LIN {X 0,Y 452.9,Z 249.571,A -85,B 0,C 180,E1 -8543.803,E2 -8543.803} C_VEL
LIN {X 0,Y 449.955,Z 249.94,A -85,B 0,C 180,E1 -8545.004,E2 -8545.004} C_VEL
LIN {X 0,Y 447.53,Z 250.24,A -85,B 0,C 180,E1 -8545.974,E2 -8545.974} C_VEL
LIN {X 0,Y 446.587,Z 250.358,A -85,B 0,C 180,E1 -8546.724,E2 -8546.724} C_VEL
LIN {X 0,Y 446.562,Z 250.36,A -85,B 0,C 180,E1 -8546.978,E2 -8546.978} C_VEL
LIN {X 0,Y 446.726,Z 250.339,A -85,B 0,C 180,E1 -8550,E2 -8550} C_VEL
LIN {X 0,Y 446.651,Z 250.351,A -85,B 0,C 180,E1 -8552.706,E2 -8552.706} C_VEL
LIN {X 0,Y 446.596,Z 250.356,A -85,B 0,C 180,E1 -8556.324,E2 -8556.324} C_VEL
LIN {X 0,Y 446.495,Z 250.369,A -85,B 0,C 180,E1 -8559.056,E2 -8559.056} C_VEL
LIN {X 0,Y 446.47,Z 250.374,A -85,B 0,C 180,E1 -8562.731,E2 -8562.731} C_VEL
LIN {X 0,Y 446.454,Z 250.374,A -85,B 0,C 180,E1 -8566.24,E2 -8566.24} C_VEL
LIN {X 0,Y 446.408,Z 250.374,A -85,B 0,C 180,E1 -8569.305,E2 -8569.305} C_VEL
LIN {X 0,Y 446.382,Z 250.382,A -85,B 0,C 180,E1 -8572.201,E2 -8572.201} C_VEL
LIN {X 0,Y 446.414,Z 250.374,A -85,B 0,C 180,E1 -8575.154,E2 -8575.154} C_VEL
LIN {X 0,Y 446.425,Z 250.378,A -85,B 0,C 180,E1 -8578.182,E2 -8578.182} C_VEL
LIN {X 0,Y 446.361,Z 250.38,A -85,B 0,C 180,E1 -8581.304,E2 -8581.304} C_VEL
LIN {X 0,Y 446.374,Z 250.381,A -85,B 0,C 180,E1 -8584.527,E2 -8584.527} C_VEL
LIN {X 0,Y 446.387,Z 250.384,A -85,B 0,C 180,E1 -8588.088,E2 -8588.088} C_VEL
LIN {X 0,Y 446.396,Z 250.376,A -85,B 0,C 180,E1 -8590.925,E2 -8590.925} C_VEL
LIN {X 0,Y 446.398,Z 250.383,A -85,B 0,C 180,E1 -8593.845,E2 -8593.845} C_VEL
LIN {X 0,Y 446.432,Z 250.373,A -85,B 0,C 180,E1 -8596.397,E2 -8596.397} C_VEL
LIN {X 0,Y 446.423,Z 250.38,A -85,B 0,C 180,E1 -8599.81,E2 -8599.81} C_VEL
LIN {X 0,Y 446.389,Z 250.379,A -85,B 0,C 180,E1 -8602.129,E2 -8602.129} C_VEL
LIN {X 0,Y 446.391,Z 250.382,A -85,B 0,C 180,E1 -8605.482,E2 -8605.482} C_VEL
LIN {X 0,Y 446.378,Z 250.378,A -85,B 0,C 180,E1 -8608.705,E2 -8608.705} C_VEL
LIN {X 0,Y 446.451,Z 250.372,A -85,B 0,C 180,E1 -8611.827,E2 -8611.827} C_VEL
LIN {X 0,Y 446.418,Z 250.375,A -85,B 0,C 180,E1 -8614.853,E2 -8614.853} C_VEL
LIN {X 0,Y 446.42,Z 250.373,A -85,B 0,C 180,E1 -8618.251,E2 -8618.251} C_VEL
LIN {X 0,Y 446.426,Z 250.374,A -85,B 0,C 180,E1 -8621.655,E2 -8621.655} C_VEL
LIN {X 0,Y 446.485,Z 250.365,A -85,B 0,C 180,E1 -8624.485,E2 -8624.485} C_VEL
LIN {X 0,Y 446.498,Z 250.363,A -85,B 0,C 180,E1 -8628.199,E2 -8628.199} C_VEL
LIN {X 0,Y 446.514,Z 250.368,A -85,B 0,C 180,E1 -8630.95,E2 -8630.95} C_VEL
LIN {X 0,Y 446.612,Z 250.349,A -85,B 0,C 180,E1 -8633.682,E2 -8633.682} C_VEL
LIN {X 0,Y 446.675,Z 250.343,A -85,B 0,C 180,E1 -8637.3,E2 -8637.3} C_VEL
LIN {X 0,Y 446.777,Z 250.329,A -85,B 0,C 180,E1 -8640.005,E2 -8640.005} C_VEL
LIN {X 0,Y 446.652,Z 250.352,A -85,B 0,C 180,E1 -8642.711,E2 -8642.711} C_VEL
LIN {X 0,Y 446.619,Z 250.352,A -85,B 0,C 180,E1 -8646.329,E2 -8646.329} C_VEL
LIN {X 0,Y 446.522,Z 250.362,A -85,B 0,C 180,E1 -8649.06,E2 -8649.06} C_VEL
LIN {X 0,Y 446.519,Z 250.364,A -85,B 0,C 180,E1 -8652.734,E2 -8652.734} C_VEL
LIN {X 0,Y 446.488,Z 250.371,A -85,B 0,C 180,E1 -8656.464,E2 -8656.464} C_VEL
LIN {X 0,Y 446.469,Z 250.367,A -85,B 0,C 180,E1 -8659.308,E2 -8659.308} C_VEL
LIN {X 0,Y 446.42,Z 250.381,A -85,B 0,C 180,E1 -8662.204,E2 -8662.204} C_VEL
LIN {X 0,Y 446.44,Z 250.37,A -85,B 0,C 180,E1 -8665.157,E2 -8665.157} C_VEL
LIN {X 0,Y 446.442,Z 250.376,A -85,B 0,C 180,E1 -8668.186,E2 -8668.186} C_VEL
LIN {X 0,Y 446.42,Z 250.373,A -85,B 0,C 180,E1 -8671.304,E2 -8671.304} C_VEL
LIN {X 0,Y 446.428,Z 250.375,A -85,B 0,C 180,E1 -8674.527,E2 -8674.527} C_VEL
LIN {X 0,Y 446.416,Z 250.38,A -85,B 0,C 180,E1 -8678.081,E2 -8678.081} C_VEL
LIN {X 0,Y 446.426,Z 250.478,A -85,B 0,C 180,E1 -8680.919,E2 -8680.919} C_VEL
LIN {X 0,Y 446.852,Z 253.496,A -85,B 0,C 180,E1 -8683.794,E2 -8683.794} C_VEL
LIN {X 0,Y 447.237,Z 256.331,A -85,B 0,C 180,E1 -8686.295,E2 -8686.295} C_VEL
LIN {X 0,Y 447.28,Z 259.62,A -85,B 0,C 180,E1 -8688.96,E2 -8688.96} C_VEL
LIN {X 0,Y 447.05,Z 263.911,A -85,B 0,C 180,E1 -8692.186,E2 -8692.186} C_VEL
LIN {X 0,Y 446.758,Z 268.648,A -85,B 0,C 180,E1 -8695.507,E2 -8695.507} C_VEL
LIN {X 0,Y 446.52,Z 272.71,A -85,B 0,C 180,E1 -8698.209,E2 -8698.209} C_VEL
LIN {X 0,Y 446.246,Z 276.741,A -85,B 0,C 180,E1 -8700.777,E2 -8700.777} C_VEL
LIN {X 0,Y 445.992,Z 281.876,A -85,B 0,C 180,E1 -8703.929,E2 -8703.929} C_VEL
LIN {X 0,Y 445.81,Z 286.721,A -85,B 0,C 180,E1 -8706.79,E2 -8706.79} C_VEL
LIN {X 0,Y 445.651,Z 291.794,A -85,B 0,C 180,E1 -8709.7,E2 -8709.7} C_VEL
LIN {X 0,Y 445.522,Z 296.887,A -85,B 0,C 180,E1 -8712.56,E2 -8712.56} C_VEL
LIN {X 0,Y 445.488,Z 299.321,A -85,B 0,C 180,E1 -8713.877,E2 -8713.877} C_VEL
LIN {X 0,Y 447.434,Z 310.041,A -85,B 0,C 180,E1 -8714.251,E2 -8714.251} C_VEL
LIN {X 0,Y 448.961,Z 320.875,A -85,B 0,C 180,E1 -8714.741,E2 -8714.741} C_VEL
LIN {X 0,Y 449.114,Z 325.65,A -85,B 0,C 180,E1 -8714.979,E2 -8714.979} C_VEL
LIN {X 0,Y 448.597,Z 336.174,A -85,B 0,C 180,E1 -8715.599,E2 -8715.599} C_VEL
LIN {X 0,Y 448.082,Z 345.452,A -85,B 0,C 180,E1 -8716.277,E2 -8716.277} C_VEL
LIN {X 0,Y 447.587,Z 354.692,A -85,B 0,C 180,E1 -8717.101,E2 -8717.101} C_VEL
LIN {X 0,Y 447.156,Z 362.932,A -85,B 0,C 180,E1 -8717.98,E2 -8717.98} C_VEL
LIN {X 0,Y 446.705,Z 370.151,A -85,B 0,C 180,E1 -8718.888,E2 -8718.888} C_VEL
LIN {X 0,Y 446.388,Z 376.355,A -85,B 0,C 180,E1 -8719.798,E2 -8719.798} C_VEL
LIN {X 0,Y 446.007,Z 382.892,A -85,B 0,C 180,E1 -8720.934,E2 -8720.934} C_VEL
LIN {X 0,Y 445.798,Z 387.393,A -85,B 0,C 180,E1 -8721.843,E2 -8721.843} C_VEL
LIN {X 0,Y 445.57,Z 393.039,A -85,B 0,C 180,E1 -8723.252,E2 -8723.252} C_VEL
LIN {X 0,Y 445.484,Z 397.207,A -85,B 0,C 180,E1 -8724.569,E2 -8724.569} C_VEL
LIN {X 0,Y 445.418,Z 399.572,A -85,B 0,C 180,E1 -8725.475,E2 -8725.475} C_VEL
LIN {X 0,Y 445.432,Z 402.755,A -85,B 0,C 180,E1 -8727.287,E2 -8727.287} C_VEL
LIN {X 0,Y 445.36,Z 403.81,A -85,B 0,C 180,E1 -8728.191,E2 -8728.191} C_VEL
LIN {X 0,Y 445.32,Z 404.396,A -85,B 0,C 180,E1 -8729.096,E2 -8729.096} C_VEL
LIN {X 0,Y 445.32,Z 404.396,A -85,B 0,C 180,E1 -8730.904,E2 -8730.904} C_VEL
LIN {X 0,Y 445.36,Z 403.81,A -85,B 0,C 180,E1 -8731.809,E2 -8731.809} C_VEL
LIN {X 0,Y 445.432,Z 402.755,A -85,B 0,C 180,E1 -8732.713,E2 -8732.713} C_VEL
LIN {X 0,Y 445.418,Z 399.572,A -85,B 0,C 180,E1 -8734.525,E2 -8734.525} C_VEL
LIN {X 0,Y 445.479,Z 395.461,A -85,B 0,C 180,E1 -8736.04,E2 -8736.04} C_VEL
LIN {X 0,Y 445.645,Z 391.224,A -85,B 0,C 180,E1 -8737.248,E2 -8737.248} C_VEL
LIN {X 0,Y 445.898,Z 385.203,A -85,B 0,C 180,E1 -8738.611,E2 -8738.611} C_VEL
LIN {X 0,Y 446.224,Z 379.107,A -85,B 0,C 180,E1 -8739.748,E2 -8739.748} C_VEL
LIN {X 0,Y 446.514,Z 373.405,A -85,B 0,C 180,E1 -8740.657,E2 -8740.657} C_VEL
LIN {X 0,Y 447.055,Z 364.852,A -85,B 0,C 180,E1 -8741.792,E2 -8741.792} C_VEL
LIN {X 0,Y 447.501,Z 356.67,A -85,B 0,C 180,E1 -8742.701,E2 -8742.701} C_VEL
LIN {X 0,Y 447.882,Z 348.534,A -85,B 0,C 180,E1 -8743.465,E2 -8743.465} C_VEL
LIN {X 0,Y 448.429,Z 339.439,A -85,B 0,C 180,E1 -8744.175,E2 -8744.175} C_VEL
LIN {X 0,Y 448.866,Z 330.686,A -85,B 0,C 180,E1 -8744.739,E2 -8744.739} C_VEL
LIN {X 0,Y 449.138,Z 322.169,A -85,B 0,C 180,E1 -8745.194,E2 -8745.194} C_VEL
LIN {X 0,Y 447.538,Z 310.77,A -85,B 0,C 180,E1 -8745.721,E2 -8745.721} C_VEL
LIN {X 0,Y 445.564,Z 300.178,A -85,B 0,C 180,E1 -8746.1,E2 -8746.1} C_VEL
LIN {X 0,Y 445.489,Z 299.318,A -85,B 0,C 180,E1 -8746.125,E2 -8746.125} C_VEL
LIN {X 0,Y 445.615,Z 293.467,A -85,B 0,C 180,E1 -8749.341,E2 -8749.341} C_VEL
LIN {X 0,Y 445.743,Z 288.39,A -85,B 0,C 180,E1 -8752.234,E2 -8752.234} C_VEL
LIN {X 0,Y 445.92,Z 283.357,A -85,B 0,C 180,E1 -8755.184,E2 -8755.184} C_VEL
LIN {X 0,Y 446.157,Z 278.379,A -85,B 0,C 180,E1 -8758.2,E2 -8758.2} C_VEL
LIN {X 0,Y 446.468,Z 273.469,A -85,B 0,C 180,E1 -8761.295,E2 -8761.295} C_VEL
LIN {X 0,Y 446.768,Z 268.64,A -85,B 0,C 180,E1 -8764.492,E2 -8764.492} C_VEL
LIN {X 0,Y 447.032,Z 263.899,A -85,B 0,C 180,E1 -8767.816,E2 -8767.816} C_VEL
LIN {X 0,Y 447.192,Z 260.798,A -85,B 0,C 180,E1 -8770.116,E2 -8770.116} C_VEL
LIN {X 0,Y 447.312,Z 257.769,A -85,B 0,C 180,E1 -8772.499,E2 -8772.499} C_VEL
LIN {X 0,Y 447.06,Z 254.794,A -85,B 0,C 180,E1 -8775.024,E2 -8775.024} C_VEL
LIN {X 0,Y 446.503,Z 250.948,A -85,B 0,C 180,E1 -8778.614,E2 -8778.614} C_VEL
LIN {X 0,Y 446.426,Z 250.477,A -85,B 0,C 180,E1 -8779.081,E2 -8779.081} C_VEL
LIN {X 0,Y 446.41,Z 250.382,A -85,B 0,C 180,E1 -8782.117,E2 -8782.117} C_VEL
LIN {X 0,Y 446.428,Z 250.378,A -85,B 0,C 180,E1 -8785.473,E2 -8785.473} C_VEL
LIN {X 0,Y 446.42,Z 250.373,A -85,B 0,C 180,E1 -8788.696,E2 -8788.696} C_VEL
LIN {X 0,Y 446.451,Z 250.375,A -85,B 0,C 180,E1 -8791.827,E2 -8791.827} C_VEL
LIN {X 0,Y 446.44,Z 250.37,A -85,B 0,C 180,E1 -8794.843,E2 -8794.843} C_VEL
LIN {X 0,Y 446.45,Z 250.371,A -85,B 0,C 180,E1 -8798.241,E2 -8798.241} C_VEL
LIN {X 0,Y 446.451,Z 250.376,A -85,B 0,C 180,E1 -8801.645,E2 -8801.645} C_VEL
LIN {X 0,Y 446.506,Z 250.362,A -85,B 0,C 180,E1 -8804.475,E2 -8804.475} C_VEL
LIN {X 0,Y 446.513,Z 250.362,A -85,B 0,C 180,E1 -8808.188,E2 -8808.188} C_VEL
LIN {X 0,Y 446.522,Z 250.362,A -85,B 0,C 180,E1 -8810.94,E2 -8810.94} C_VEL
LIN {X 0,Y 446.619,Z 250.352,A -85,B 0,C 180,E1 -8813.671,E2 -8813.671} C_VEL
LIN {X 0,Y 446.652,Z 250.352,A -85,B 0,C 180,E1 -8817.289,E2 -8817.289} C_VEL
LIN {X 0,Y 446.777,Z 250.329,A -85,B 0,C 180,E1 -8819.995,E2 -8819.995} C_VEL
LIN {X 0,Y 446.675,Z 250.343,A -85,B 0,C 180,E1 -8822.7,E2 -8822.7} C_VEL
LIN {X 0,Y 446.612,Z 250.349,A -85,B 0,C 180,E1 -8826.318,E2 -8826.318} C_VEL
LIN {X 0,Y 446.514,Z 250.368,A -85,B 0,C 180,E1 -8829.05,E2 -8829.05} C_VEL
LIN {X 0,Y 446.501,Z 250.368,A -85,B 0,C 180,E1 -8832.724,E2 -8832.724} C_VEL
LIN {X 0,Y 446.472,Z 250.367,A -85,B 0,C 180,E1 -8836.222,E2 -8836.222} C_VEL
LIN {X 0,Y 446.442,Z 250.372,A -85,B 0,C 180,E1 -8839.298,E2 -8839.298} C_VEL
LIN {X 0,Y 446.389,Z 250.379,A -85,B 0,C 180,E1 -8842.194,E2 -8842.194} C_VEL
LIN {X 0,Y 446.418,Z 250.375,A -85,B 0,C 180,E1 -8845.147,E2 -8845.147} C_VEL
LIN {X 0,Y 446.451,Z 250.372,A -85,B 0,C 180,E1 -8848.173,E2 -8848.173} C_VEL
LIN {X 0,Y 446.381,Z 250.378,A -85,B 0,C 180,E1 -8851.769,E2 -8851.769} C_VEL
LIN {X 0,Y 446.391,Z 250.382,A -85,B 0,C 180,E1 -8854.518,E2 -8854.518} C_VEL
LIN {X 0,Y 446.392,Z 250.381,A -85,B 0,C 180,E1 -8858.077,E2 -8858.077} C_VEL
LIN {X 0,Y 446.403,Z 250.376,A -85,B 0,C 180,E1 -8860.916,E2 -8860.916} C_VEL
LIN {X 0,Y 446.432,Z 250.375,A -85,B 0,C 180,E1 -8863.831,E2 -8863.831} C_VEL
LIN {X 0,Y 446.4,Z 250.376,A -85,B 0,C 180,E1 -8867.393,E2 -8867.393} C_VEL
LIN {X 0,Y 446.444,Z 250.372,A -85,B 0,C 180,E1 -8870.464,E2 -8870.464} C_VEL
LIN {X 0,Y 446.353,Z 250.383,A -85,B 0,C 180,E1 -8873.405,E2 -8873.405} C_VEL
LIN {X 0,Y 446.392,Z 250.377,A -85,B 0,C 180,E1 -8876.563,E2 -8876.563} C_VEL
LIN {X 0,Y 446.382,Z 250.382,A -85,B 0,C 180,E1 -8879.973,E2 -8879.973} C_VEL
LIN {X 0,Y 446.422,Z 250.373,A -85,B 0,C 180,E1 -8882.836,E2 -8882.836} C_VEL
LIN {X 0,Y 446.411,Z 250.378,A -85,B 0,C 180,E1 -8885.918,E2 -8885.918} C_VEL
LIN {X 0,Y 446.433,Z 250.372,A -85,B 0,C 180,E1 -8888.773,E2 -8888.773} C_VEL
LIN {X 0,Y 446.401,Z 250.382,A -85,B 0,C 180,E1 -8891.647,E2 -8891.647} C_VEL
LIN {X 0,Y 446.462,Z 250.371,A -85,B 0,C 180,E1 -8894.479,E2 -8894.479} C_VEL
LIN {X 0,Y 446.481,Z 250.368,A -85,B 0,C 180,E1 -8898.192,E2 -8898.192} C_VEL
LIN {X 0,Y 446.54,Z 250.362,A -85,B 0,C 180,E1 -8901.857,E2 -8901.857} C_VEL
LIN {X 0,Y 446.591,Z 250.356,A -85,B 0,C 180,E1 -8904.582,E2 -8904.582} C_VEL
LIN {X 0,Y 446.562,Z 250.36,A -85,B 0,C 180,E1 -8906.978,E2 -8906.978} C_VEL
LIN {X 0,Y 446.044,Z 250.428,A -85,B 0,C 180,E1 -8907.731,E2 -8907.731} C_VEL
LIN {X 0,Y 443.253,Z 250.781,A -85,B 0,C 180,E1 -8908.955,E2 -8908.955} C_VEL
LIN {X 0,Y 440.784,Z 251.087,A -85,B 0,C 180,E1 -8909.942,E2 -8909.942} C_VEL
LIN {X 0,Y 439.689,Z 251.219,A -85,B 0,C 180,E1 -8910.705,E2 -8910.705} C_VEL
LIN {X 0,Y 439.587,Z 251.23,A -85,B 0,C 180,E1 -8910.964,E2 -8910.964} C_VEL
LIN {X 0,Y 439.599,Z 251.229,A -85,B 0,C 180,E1 -8912.749,E2 -8912.749} C_VEL
LIN {X 0,Y 439.566,Z 251.233,A -85,B 0,C 180,E1 -8916.426,E2 -8916.426} C_VEL
LIN {X 0,Y 439.452,Z 251.246,A -85,B 0,C 180,E1 -8919.202,E2 -8919.202} C_VEL
LIN {X 0,Y 439.439,Z 251.25,A -85,B 0,C 180,E1 -8922.728,E2 -8922.728} C_VEL
LIN {X 0,Y 439.397,Z 251.254,A -85,B 0,C 180,E1 -8926.357,E2 -8926.357} C_VEL
LIN {X 0,Y 439.373,Z 251.252,A -85,B 0,C 180,E1 -8929.627,E2 -8929.627} C_VEL
LIN {X 0,Y 439.324,Z 251.263,A -85,B 0,C 180,E1 -8932.577,E2 -8932.577} C_VEL
LIN {X 0,Y 439.354,Z 251.253,A -85,B 0,C 180,E1 -8935.587,E2 -8935.587} C_VEL
LIN {X 0,Y 439.366,Z 251.254,A -85,B 0,C 180,E1 -8938.676,E2 -8938.676} C_VEL
LIN {X 0,Y 439.316,Z 251.261,A -85,B 0,C 180,E1 -8941.864,E2 -8941.864} C_VEL
LIN {X 0,Y 439.345,Z 251.254,A -85,B 0,C 180,E1 -8945.16,E2 -8945.16} C_VEL
LIN {X 0,Y 439.349,Z 251.255,A -85,B 0,C 180,E1 -8948.597,E2 -8948.597} C_VEL
LIN {X 0,Y 439.354,Z 251.254,A -85,B 0,C 180,E1 -8951.264,E2 -8951.264} C_VEL
LIN {X 0,Y 439.368,Z 251.251,A -85,B 0,C 180,E1 -8954.732,E2 -8954.732} C_VEL
LIN {X 0,Y 439.369,Z 251.259,A -85,B 0,C 180,E1 -8957.803,E2 -8957.803} C_VEL
LIN {X 0,Y 439.405,Z 251.249,A -85,B 0,C 180,E1 -8960.235,E2 -8960.235} C_VEL
LIN {X 0,Y 439.336,Z 251.262,A -85,B 0,C 180,E1 -8963.718,E2 -8963.718} C_VEL
LIN {X 0,Y 439.334,Z 251.257,A -85,B 0,C 180,E1 -8967.059,E2 -8967.059} C_VEL
LIN {X 0,Y 439.346,Z 251.254,A -85,B 0,C 180,E1 -8970.28,E2 -8970.28} C_VEL
LIN {X 0,Y 439.396,Z 251.255,A -85,B 0,C 180,E1 -8973.402,E2 -8973.402} C_VEL
LIN {X 0,Y 439.356,Z 251.253,A -85,B 0,C 180,E1 -8976.435,E2 -8976.435} C_VEL
LIN {X 0,Y 439.361,Z 251.258,A -85,B 0,C 180,E1 -8979.403,E2 -8979.403} C_VEL
LIN {X 0,Y 439.38,Z 251.25,A -85,B 0,C 180,E1 -8982.314,E2 -8982.314} C_VEL
LIN {X 0,Y 439.425,Z 251.251,A -85,B 0,C 180,E1 -8985.18,E2 -8985.18} C_VEL
LIN {X 0,Y 439.464,Z 251.239,A -85,B 0,C 180,E1 -8988.007,E2 -8988.007} C_VEL
LIN {X 0,Y 439.487,Z 251.237,A -85,B 0,C 180,E1 -8991.731,E2 -8991.731} C_VEL
LIN {X 0,Y 439.594,Z 251.226,A -85,B 0,C 180,E1 -8994.501,E2 -8994.501} C_VEL
LIN {X 0,Y 439.622,Z 251.221,A -85,B 0,C 180,E1 -8998.173,E2 -8998.173} C_VEL
LIN {X 0,Y 439.747,Z 251.204,A -85,B 0,C 180,E1 -9000.005,E2 -9000.005} C_VEL
LIN {X 0,Y 439.603,Z 251.229,A -85,B 0,C 180,E1 -9002.754,E2 -9002.754} C_VEL
LIN {X 0,Y 439.59,Z 251.229,A -85,B 0,C 180,E1 -9006.431,E2 -9006.431} C_VEL
LIN {X 0,Y 439.486,Z 251.237,A -85,B 0,C 180,E1 -9009.207,E2 -9009.207} C_VEL
LIN {X 0,Y 439.463,Z 251.241,A -85,B 0,C 180,E1 -9012.942,E2 -9012.942} C_VEL
LIN {X 0,Y 439.445,Z 251.249,A -85,B 0,C 180,E1 -9016.352,E2 -9016.352} C_VEL
LIN {X 0,Y 439.403,Z 251.248,A -85,B 0,C 180,E1 -9019.631,E2 -9019.631} C_VEL
LIN {X 0,Y 439.365,Z 251.255,A -85,B 0,C 180,E1 -9022.58,E2 -9022.58} C_VEL
LIN {X 0,Y 439.378,Z 251.252,A -85,B 0,C 180,E1 -9025.591,E2 -9025.591} C_VEL
LIN {X 0,Y 439.395,Z 251.249,A -85,B 0,C 180,E1 -9028.679,E2 -9028.679} C_VEL
LIN {X 0,Y 439.374,Z 251.257,A -85,B 0,C 180,E1 -9032.033,E2 -9032.033} C_VEL
LIN {X 0,Y 439.396,Z 251.249,A -85,B 0,C 180,E1 -9035.343,E2 -9035.343} C_VEL
LIN {X 0,Y 439.368,Z 251.257,A -85,B 0,C 180,E1 -9038.601,E2 -9038.601} C_VEL
LIN {X 0,Y 439.354,Z 251.26,A -85,B 0,C 180,E1 -9039.843,E2 -9039.843} C_VEL
LIN {X 0,Y 439.491,Z 252.002,A -85,B 0,C 180,E1 -9041.274,E2 -9041.274} C_VEL
LIN {X 0,Y 439.893,Z 254.89,A -85,B 0,C 180,E1 -9044.034,E2 -9044.034} C_VEL
LIN {X 0,Y 440.24,Z 257.847,A -85,B 0,C 180,E1 -9046.651,E2 -9046.651} C_VEL
LIN {X 0,Y 440.236,Z 260.851,A -85,B 0,C 180,E1 -9049.117,E2 -9049.117} C_VEL
LIN {X 0,Y 440.095,Z 263.955,A -85,B 0,C 180,E1 -9051.494,E2 -9051.494} C_VEL
LIN {X 0,Y 439.775,Z 268.634,A -85,B 0,C 180,E1 -9054.88,E2 -9054.88} C_VEL
LIN {X 0,Y 439.476,Z 273.44,A -85,B 0,C 180,E1 -9058.149,E2 -9058.149} C_VEL
LIN {X 0,Y 439.122,Z 278.32,A -85,B 0,C 180,E1 -9061.306,E2 -9061.306} C_VEL
LIN {X 0,Y 438.876,Z 283.271,A -85,B 0,C 180,E1 -9064.383,E2 -9064.383} C_VEL
LIN {X 0,Y 438.677,Z 288.279,A -85,B 0,C 180,E1 -9067.388,E2 -9067.388} C_VEL
LIN {X 0,Y 438.544,Z 293.332,A -85,B 0,C 180,E1 -9070.334,E2 -9070.334} C_VEL
LIN {X 0,Y 438.414,Z 299.15,A -85,B 0,C 180,E1 -9073.608,E2 -9073.608} C_VEL
LIN {X 0,Y 440.551,Z 310.914,A -85,B 0,C 180,E1 -9074.035,E2 -9074.035} C_VEL
LIN {X 0,Y 442.279,Z 323.261,A -85,B 0,C 180,E1 -9074.623,E2 -9074.623} C_VEL
LIN {X 0,Y 441.708,Z 335.979,A -85,B 0,C 180,E1 -9075.37,E2 -9075.37} C_VEL
LIN {X 0,Y 441.176,Z 345.257,A -85,B 0,C 180,E1 -9076.058,E2 -9076.058} C_VEL
LIN {X 0,Y 440.752,Z 353.31,A -85,B 0,C 180,E1 -9076.774,E2 -9076.774} C_VEL
LIN {X 0,Y 440.316,Z 360.817,A -85,B 0,C 180,E1 -9077.557,E2 -9077.557} C_VEL
LIN {X 0,Y 439.723,Z 369.956,A -85,B 0,C 180,E1 -9078.709,E2 -9078.709} C_VEL
LIN {X 0,Y 439.364,Z 376.159,A -85,B 0,C 180,E1 -9079.633,E2 -9079.633} C_VEL
LIN {X 0,Y 438.981,Z 382.697,A -85,B 0,C 180,E1 -9080.788,E2 -9080.788} C_VEL
LIN {X 0,Y 438.751,Z 387.198,A -85,B 0,C 180,E1 -9081.711,E2 -9081.711} C_VEL
LIN {X 0,Y 438.512,Z 392.689,A -85,B 0,C 180,E1 -9083.096,E2 -9083.096} C_VEL
LIN {X 0,Y 438.383,Z 397.012,A -85,B 0,C 180,E1 -9084.48,E2 -9084.48} C_VEL
LIN {X 0,Y 438.348,Z 399.377,A -85,B 0,C 180,E1 -9085.402,E2 -9085.402} C_VEL
LIN {X 0,Y 438.265,Z 401.173,A -85,B 0,C 180,E1 -9086.322,E2 -9086.322} C_VEL
LIN {X 0,Y 438.34,Z 402.561,A -85,B 0,C 180,E1 -9087.243,E2 -9087.243} C_VEL
LIN {X 0,Y 438.283,Z 403.616,A -85,B 0,C 180,E1 -9088.162,E2 -9088.162} C_VEL
LIN {X 0,Y 438.235,Z 404.202,A -85,B 0,C 180,E1 -9089.081,E2 -9089.081} C_VEL
LIN {X 0,Y 438.235,Z 404.202,A -85,B 0,C 180,E1 -9090.919,E2 -9090.919} C_VEL
LIN {X 0,Y 438.283,Z 403.616,A -85,B 0,C 180,E1 -9091.838,E2 -9091.838} C_VEL
LIN {X 0,Y 438.34,Z 402.561,A -85,B 0,C 180,E1 -9092.757,E2 -9092.757} C_VEL
LIN {X 0,Y 438.265,Z 401.173,A -85,B 0,C 180,E1 -9093.678,E2 -9093.678} C_VEL
LIN {X 0,Y 438.389,Z 398.229,A -85,B 0,C 180,E1 -9095.058,E2 -9095.058} C_VEL
LIN {X 0,Y 438.46,Z 394.242,A -85,B 0,C 180,E1 -9096.442,E2 -9096.442} C_VEL
LIN {X 0,Y 438.661,Z 389.114,A -85,B 0,C 180,E1 -9097.827,E2 -9097.827} C_VEL
LIN {X 0,Y 438.9,Z 383.852,A -85,B 0,C 180,E1 -9098.982,E2 -9098.982} C_VEL
LIN {X 0,Y 439.279,Z 377.535,A -85,B 0,C 180,E1 -9100.136,E2 -9100.136} C_VEL
LIN {X 0,Y 439.596,Z 371.583,A -85,B 0,C 180,E1 -9101.06,E2 -9101.06} C_VEL
LIN {X 0,Y 440.078,Z 364.656,A -85,B 0,C 180,E1 -9101.982,E2 -9101.982} C_VEL
LIN {X 0,Y 440.54,Z 356.474,A -85,B 0,C 180,E1 -9102.905,E2 -9102.905} C_VEL
LIN {X 0,Y 440.981,Z 347.693,A -85,B 0,C 180,E1 -9103.736,E2 -9103.736} C_VEL
LIN {X 0,Y 441.506,Z 339.243,A -85,B 0,C 180,E1 -9104.402,E2 -9104.402} C_VEL
LIN {X 0,Y 442.003,Z 330.491,A -85,B 0,C 180,E1 -9104.974,E2 -9104.974} C_VEL
LIN {X 0,Y 442.287,Z 323.262,A -85,B 0,C 180,E1 -9105.376,E2 -9105.376} C_VEL
LIN {X 0,Y 440.606,Z 311.162,A -85,B 0,C 180,E1 -9105.955,E2 -9105.955} C_VEL
LIN {X 0,Y 438.534,Z 300.22,A -85,B 0,C 180,E1 -9106.359,E2 -9106.359} C_VEL
LIN {X 0,Y 438.413,Z 299.149,A -85,B 0,C 180,E1 -9106.393,E2 -9106.393} C_VEL
LIN {X 0,Y 438.543,Z 293.33,A -85,B 0,C 180,E1 -9109.666,E2 -9109.666} C_VEL
LIN {X 0,Y 438.692,Z 288.278,A -85,B 0,C 180,E1 -9112.611,E2 -9112.611} C_VEL
LIN {X 0,Y 438.88,Z 283.27,A -85,B 0,C 180,E1 -9115.617,E2 -9115.617} C_VEL
LIN {X 0,Y 439.121,Z 278.317,A -85,B 0,C 180,E1 -9118.694,E2 -9118.694} C_VEL
LIN {X 0,Y 439.486,Z 273.434,A -85,B 0,C 180,E1 -9121.85,E2 -9121.85} C_VEL
LIN {X 0,Y 439.788,Z 268.625,A -85,B 0,C 180,E1 -9125.119,E2 -9125.119} C_VEL
LIN {X 0,Y 440.072,Z 263.921,A -85,B 0,C 180,E1 -9128.522,E2 -9128.522} C_VEL
LIN {X 0,Y 440.284,Z 260.209,A -85,B 0,C 180,E1 -9131.385,E2 -9131.385} C_VEL
LIN {X 0,Y 440.16,Z 256.981,A -85,B 0,C 180,E1 -9134.064,E2 -9134.064} C_VEL
LIN {X 0,Y 439.71,Z 253.437,A -85,B 0,C 180,E1 -9137.325,E2 -9137.325} C_VEL
LIN {X 0,Y 439.453,Z 251.708,A -85,B 0,C 180,E1 -9139.023,E2 -9139.023} C_VEL
LIN {X 0,Y 439.367,Z 251.258,A -85,B 0,C 180,E1 -9140.217,E2 -9140.217} C_VEL
LIN {X 0,Y 439.377,Z 251.256,A -85,B 0,C 180,E1 -9143.709,E2 -9143.709} C_VEL
LIN {X 0,Y 439.377,Z 251.25,A -85,B 0,C 180,E1 -9147.05,E2 -9147.05} C_VEL
LIN {X 0,Y 439.377,Z 251.254,A -85,B 0,C 180,E1 -9150.27,E2 -9150.27} C_VEL
LIN {X 0,Y 439.373,Z 251.252,A -85,B 0,C 180,E1 -9153.388,E2 -9153.388} C_VEL
LIN {X 0,Y 439.384,Z 251.25,A -85,B 0,C 180,E1 -9156.425,E2 -9156.425} C_VEL
LIN {X 0,Y 439.388,Z 251.252,A -85,B 0,C 180,E1 -9159.393,E2 -9159.393} C_VEL
LIN {X 0,Y 439.403,Z 251.248,A -85,B 0,C 180,E1 -9162.304,E2 -9162.304} C_VEL
LIN {X 0,Y 439.445,Z 251.244,A -85,B 0,C 180,E1 -9165.169,E2 -9165.169} C_VEL
LIN {X 0,Y 439.48,Z 251.24,A -85,B 0,C 180,E1 -9167.996,E2 -9167.996} C_VEL
LIN {X 0,Y 439.497,Z 251.239,A -85,B 0,C 180,E1 -9171.72,E2 -9171.72} C_VEL
LIN {X 0,Y 439.602,Z 251.222,A -85,B 0,C 180,E1 -9174.491,E2 -9174.491} C_VEL
LIN {X 0,Y 439.617,Z 251.22,A -85,B 0,C 180,E1 -9178.163,E2 -9178.163} C_VEL
LIN {X 0,Y 439.747,Z 251.204,A -85,B 0,C 180,E1 -9179.995,E2 -9179.995} C_VEL
LIN {X 0,Y 439.625,Z 251.222,A -85,B 0,C 180,E1 -9182.743,E2 -9182.743} C_VEL
LIN {X 0,Y 439.583,Z 251.225,A -85,B 0,C 180,E1 -9186.42,E2 -9186.42} C_VEL
LIN {X 0,Y 439.477,Z 251.243,A -85,B 0,C 180,E1 -9189.196,E2 -9189.196} C_VEL
LIN {X 0,Y 439.445,Z 251.249,A -85,B 0,C 180,E1 -9192.932,E2 -9192.932} C_VEL
LIN {X 0,Y 439.423,Z 251.246,A -85,B 0,C 180,E1 -9196.342,E2 -9196.342} C_VEL
LIN {X 0,Y 439.376,Z 251.25,A -85,B 0,C 180,E1 -9199.621,E2 -9199.621} C_VEL
LIN {X 0,Y 439.336,Z 251.262,A -85,B 0,C 180,E1 -9202.57,E2 -9202.57} C_VEL
LIN {X 0,Y 439.369,Z 251.251,A -85,B 0,C 180,E1 -9205.58,E2 -9205.58} C_VEL
LIN {X 0,Y 439.383,Z 251.255,A -85,B 0,C 180,E1 -9208.668,E2 -9208.668} C_VEL
LIN {X 0,Y 439.332,Z 251.258,A -85,B 0,C 180,E1 -9212.025,E2 -9212.025} C_VEL
LIN {X 0,Y 439.356,Z 251.253,A -85,B 0,C 180,E1 -9215.335,E2 -9215.335} C_VEL
LIN {X 0,Y 439.352,Z 251.257,A -85,B 0,C 180,E1 -9218.588,E2 -9218.588} C_VEL
LIN {X 0,Y 439.36,Z 251.252,A -85,B 0,C 180,E1 -9221.254,E2 -9221.254} C_VEL
LIN {X 0,Y 439.394,Z 251.249,A -85,B 0,C 180,E1 -9224.719,E2 -9224.719} C_VEL
LIN {X 0,Y 439.362,Z 251.256,A -85,B 0,C 180,E1 -9227.793,E2 -9227.793} C_VEL
LIN {X 0,Y 439.403,Z 251.251,A -85,B 0,C 180,E1 -9230.226,E2 -9230.226} C_VEL
LIN {X 0,Y 439.322,Z 251.262,A -85,B 0,C 180,E1 -9233.709,E2 -9233.709} C_VEL
LIN {X 0,Y 439.316,Z 251.258,A -85,B 0,C 180,E1 -9237.05,E2 -9237.05} C_VEL
LIN {X 0,Y 439.337,Z 251.257,A -85,B 0,C 180,E1 -9240.272,E2 -9240.272} C_VEL
LIN {X 0,Y 439.37,Z 251.255,A -85,B 0,C 180,E1 -9243.393,E2 -9243.393} C_VEL
LIN {X 0,Y 439.339,Z 251.255,A -85,B 0,C 180,E1 -9246.427,E2 -9246.427} C_VEL
LIN {X 0,Y 439.351,Z 251.26,A -85,B 0,C 180,E1 -9249.396,E2 -9249.396} C_VEL
LIN {X 0,Y 439.375,Z 251.254,A -85,B 0,C 180,E1 -9252.308,E2 -9252.308} C_VEL
LIN {X 0,Y 439.399,Z 251.254,A -85,B 0,C 180,E1 -9255.173,E2 -9255.173} C_VEL
LIN {X 0,Y 439.447,Z 251.244,A -85,B 0,C 180,E1 -9258.001,E2 -9258.001} C_VEL
LIN {X 0,Y 439.488,Z 251.241,A -85,B 0,C 180,E1 -9261.725,E2 -9261.725} C_VEL
LIN {X 0,Y 439.566,Z 251.231,A -85,B 0,C 180,E1 -9264.495,E2 -9264.495} C_VEL
LIN {X 0,Y 439.57,Z 251.229,A -85,B 0,C 180,E1 -9268.168,E2 -9268.168} C_VEL
LIN {X 0,Y 439.697,Z 251.215,A -85,B 0,C 180,E1 -9270,E2 -9270} C_VEL
LIN {X 0,Y 439.587,Z 251.23,A -85,B 0,C 180,E1 -9270.964,E2 -9270.964} C_VEL
LIN {X 0,Y 438.85,Z 251.319,A -85,B 0,C 180,E1 -9271.728,E2 -9271.728} C_VEL
LIN {X 0,Y 435.861,Z 251.694,A -85,B 0,C 180,E1 -9272.967,E2 -9272.967} C_VEL
LIN {X 0,Y 433.413,Z 251.999,A -85,B 0,C 180,E1 -9273.967,E2 -9273.967} C_VEL
LIN {X 0,Y 432.442,Z 252.12,A -85,B 0,C 180,E1 -9274.742,E2 -9274.742} C_VEL
LIN {X 0,Y 432.404,Z 252.122,A -85,B 0,C 180,E1 -9275.004,E2 -9275.004} C_VEL
LIN {X 0,Y 432.52,Z 252.109,A -85,B 0,C 180,E1 -9277.68,E2 -9277.68} C_VEL
LIN {X 0,Y 432.35,Z 252.13,A -85,B 0,C 180,E1 -9281.248,E2 -9281.248} C_VEL
LIN {X 0,Y 432.329,Z 252.133,A -85,B 0,C 180,E1 -9284.113,E2 -9284.113} C_VEL
LIN {X 0,Y 432.338,Z 252.133,A -85,B 0,C 180,E1 -9287.014,E2 -9287.014} C_VEL
LIN {X 0,Y 432.32,Z 252.134,A -85,B 0,C 180,E1 -9289.961,E2 -9289.961} C_VEL
LIN {X 0,Y 432.273,Z 252.137,A -85,B 0,C 180,E1 -9292.966,E2 -9292.966} C_VEL
LIN {X 0,Y 432.309,Z 252.134,A -85,B 0,C 180,E1 -9296.035,E2 -9296.035} C_VEL
LIN {X 0,Y 432.294,Z 252.133,A -85,B 0,C 180,E1 -9299.19,E2 -9299.19} C_VEL
LIN {X 0,Y 432.268,Z 252.142,A -85,B 0,C 180,E1 -9302.297,E2 -9302.297} C_VEL
LIN {X 0,Y 432.285,Z 252.135,A -85,B 0,C 180,E1 -9304.681,E2 -9304.681} C_VEL
LIN {X 0,Y 432.302,Z 252.138,A -85,B 0,C 180,E1 -9308.152,E2 -9308.152} C_VEL
LIN {X 0,Y 432.323,Z 252.132,A -85,B 0,C 180,E1 -9311.613,E2 -9311.613} C_VEL
LIN {X 0,Y 432.331,Z 252.13,A -85,B 0,C 180,E1 -9314.346,E2 -9314.346} C_VEL
LIN {X 0,Y 432.327,Z 252.129,A -85,B 0,C 180,E1 -9317.013,E2 -9317.013} C_VEL
LIN {X 0,Y 432.313,Z 252.137,A -85,B 0,C 180,E1 -9319.822,E2 -9319.822} C_VEL
LIN {X 0,Y 432.275,Z 252.136,A -85,B 0,C 180,E1 -9323.028,E2 -9323.028} C_VEL
LIN {X 0,Y 432.321,Z 252.132,A -85,B 0,C 180,E1 -9326.002,E2 -9326.002} C_VEL
LIN {X 0,Y 432.311,Z 252.138,A -85,B 0,C 180,E1 -9329.496,E2 -9329.496} C_VEL
LIN {X 0,Y 432.358,Z 252.126,A -85,B 0,C 180,E1 -9332.934,E2 -9332.934} C_VEL
LIN {X 0,Y 432.34,Z 252.128,A -85,B 0,C 180,E1 -9336.029,E2 -9336.029} C_VEL
LIN {X 0,Y 432.323,Z 252.133,A -85,B 0,C 180,E1 -9339.052,E2 -9339.052} C_VEL
LIN {X 0,Y 432.336,Z 252.128,A -85,B 0,C 180,E1 -9342.016,E2 -9342.016} C_VEL
LIN {X 0,Y 432.372,Z 252.128,A -85,B 0,C 180,E1 -9344.932,E2 -9344.932} C_VEL
LIN {X 0,Y 432.439,Z 252.115,A -85,B 0,C 180,E1 -9347.809,E2 -9347.809} C_VEL
LIN {X 0,Y 432.447,Z 252.114,A -85,B 0,C 180,E1 -9351.595,E2 -9351.595} C_VEL
LIN {X 0,Y 432.571,Z 252.1,A -85,B 0,C 180,E1 -9354.412,E2 -9354.412} C_VEL
LIN {X 0,Y 432.592,Z 252.096,A -85,B 0,C 180,E1 -9358.144,E2 -9358.144} C_VEL
LIN {X 0,Y 432.717,Z 252.08,A -85,B 0,C 180,E1 -9360.005,E2 -9360.005} C_VEL
LIN {X 0,Y 432.557,Z 252.106,A -85,B 0,C 180,E1 -9362.799,E2 -9362.799} C_VEL
LIN {X 0,Y 432.578,Z 252.097,A -85,B 0,C 180,E1 -9365.599,E2 -9365.599} C_VEL
LIN {X 0,Y 432.457,Z 252.118,A -85,B 0,C 180,E1 -9368.415,E2 -9368.415} C_VEL
LIN {X 0,Y 432.456,Z 252.117,A -85,B 0,C 180,E1 -9372.201,E2 -9372.201} C_VEL
LIN {X 0,Y 432.429,Z 252.119,A -85,B 0,C 180,E1 -9376.044,E2 -9376.044} C_VEL
LIN {X 0,Y 432.388,Z 252.121,A -85,B 0,C 180,E1 -9379.489,E2 -9379.489} C_VEL
LIN {X 0,Y 432.319,Z 252.13,A -85,B 0,C 180,E1 -9382.969,E2 -9382.969} C_VEL
LIN {X 0,Y 432.339,Z 252.127,A -85,B 0,C 180,E1 -9385.006,E2 -9385.006} C_VEL
LIN {X 0,Y 432.352,Z 252.127,A -85,B 0,C 180,E1 -9388.626,E2 -9388.626} C_VEL
LIN {X 0,Y 432.325,Z 252.13,A -85,B 0,C 180,E1 -9391.35,E2 -9391.35} C_VEL
LIN {X 0,Y 432.34,Z 252.129,A -85,B 0,C 180,E1 -9394.681,E2 -9394.681} C_VEL
LIN {X 0,Y 432.336,Z 252.134,A -85,B 0,C 180,E1 -9398.154,E2 -9398.154} C_VEL
LIN {X 0,Y 432.317,Z 252.137,A -85,B 0,C 180,E1 -9400.178,E2 -9400.178} C_VEL
LIN {X 0,Y 432.739,Z 254.967,A -85,B 0,C 180,E1 -9403.045,E2 -9403.045} C_VEL
LIN {X 0,Y 433.114,Z 257.899,A -85,B 0,C 180,E1 -9405.755,E2 -9405.755} C_VEL
LIN {X 0,Y 433.266,Z 260.903,A -85,B 0,C 180,E1 -9408.314,E2 -9408.314} C_VEL
LIN {X 0,Y 433.077,Z 264.514,A -85,B 0,C 180,E1 -9411.169,E2 -9411.169} C_VEL
LIN {X 0,Y 432.784,Z 268.72,A -85,B 0,C 180,E1 -9414.291,E2 -9414.291} C_VEL
LIN {X 0,Y 432.468,Z 273.562,A -85,B 0,C 180,E1 -9417.682,E2 -9417.682} C_VEL
LIN {X 0,Y 432.101,Z 278.26,A -85,B 0,C 180,E1 -9420.795,E2 -9420.795} C_VEL
LIN {X 0,Y 431.853,Z 283.184,A -85,B 0,C 180,E1 -9423.935,E2 -9423.935} C_VEL
LIN {X 0,Y 431.641,Z 288.166,A -85,B 0,C 180,E1 -9426.998,E2 -9426.998} C_VEL
LIN {X 0,Y 431.468,Z 293.195,A -85,B 0,C 180,E1 -9429.998,E2 -9429.998} C_VEL
LIN {X 0,Y 431.345,Z 298.962,A -85,B 0,C 180,E1 -9433.33,E2 -9433.33} C_VEL
LIN {X 0,Y 433.38,Z 310.157,A -85,B 0,C 180,E1 -9433.744,E2 -9433.744} C_VEL
LIN {X 0,Y 434.894,Z 320.475,A -85,B 0,C 180,E1 -9434.235,E2 -9434.235} C_VEL
LIN {X 0,Y 435.403,Z 325.26,A -85,B 0,C 180,E1 -9434.494,E2 -9434.494} C_VEL
LIN {X 0,Y 434.82,Z 335.784,A -85,B 0,C 180,E1 -9435.133,E2 -9435.133} C_VEL
LIN {X 0,Y 434.276,Z 345.062,A -85,B 0,C 180,E1 -9435.832,E2 -9435.832} C_VEL
LIN {X 0,Y 433.775,Z 353.889,A -85,B 0,C 180,E1 -9436.639,E2 -9436.639} C_VEL
LIN {X 0,Y 433.237,Z 362.541,A -85,B 0,C 180,E1 -9437.588,E2 -9437.588} C_VEL
LIN {X 0,Y 432.752,Z 369.761,A -85,B 0,C 180,E1 -9438.525,E2 -9438.525} C_VEL
LIN {X 0,Y 432.342,Z 375.963,A -85,B 0,C 180,E1 -9439.463,E2 -9439.463} C_VEL
LIN {X 0,Y 431.93,Z 382.501,A -85,B 0,C 180,E1 -9440.636,E2 -9440.636} C_VEL
LIN {X 0,Y 431.692,Z 387.003,A -85,B 0,C 180,E1 -9441.575,E2 -9441.575} C_VEL
LIN {X 0,Y 431.436,Z 392.493,A -85,B 0,C 180,E1 -9442.983,E2 -9442.983} C_VEL
LIN {X 0,Y 431.286,Z 396.816,A -85,B 0,C 180,E1 -9444.389,E2 -9444.389} C_VEL
LIN {X 0,Y 431.277,Z 399.183,A -85,B 0,C 180,E1 -9445.327,E2 -9445.327} C_VEL
LIN {X 0,Y 431.174,Z 400.978,A -85,B 0,C 180,E1 -9446.262,E2 -9446.262} C_VEL
LIN {X 0,Y 431.208,Z 403.422,A -85,B 0,C 180,E1 -9448.132,E2 -9448.132} C_VEL
LIN {X 0,Y 431.154,Z 404.008,A -85,B 0,C 180,E1 -9449.066,E2 -9449.066} C_VEL
LIN {X 0,Y 431.154,Z 404.008,A -85,B 0,C 180,E1 -9450.934,E2 -9450.934} C_VEL
LIN {X 0,Y 431.208,Z 403.422,A -85,B 0,C 180,E1 -9451.868,E2 -9451.868} C_VEL
LIN {X 0,Y 431.174,Z 400.978,A -85,B 0,C 180,E1 -9453.738,E2 -9453.738} C_VEL
LIN {X 0,Y 431.3,Z 398.034,A -85,B 0,C 180,E1 -9455.142,E2 -9455.142} C_VEL
LIN {X 0,Y 431.389,Z 394.047,A -85,B 0,C 180,E1 -9456.548,E2 -9456.548} C_VEL
LIN {X 0,Y 431.588,Z 388.918,A -85,B 0,C 180,E1 -9457.956,E2 -9457.956} C_VEL
LIN {X 0,Y 431.851,Z 383.656,A -85,B 0,C 180,E1 -9459.13,E2 -9459.13} C_VEL
LIN {X 0,Y 432.244,Z 377.339,A -85,B 0,C 180,E1 -9460.303,E2 -9460.303} C_VEL
LIN {X 0,Y 432.612,Z 371.387,A -85,B 0,C 180,E1 -9461.241,E2 -9461.241} C_VEL
LIN {X 0,Y 433.115,Z 364.461,A -85,B 0,C 180,E1 -9462.178,E2 -9462.178} C_VEL
LIN {X 0,Y 433.591,Z 356.279,A -85,B 0,C 180,E1 -9463.116,E2 -9463.116} C_VEL
LIN {X 0,Y 434.067,Z 347.415,A -85,B 0,C 180,E1 -9463.967,E2 -9463.967} C_VEL
LIN {X 0,Y 434.619,Z 339.048,A -85,B 0,C 180,E1 -9464.635,E2 -9464.635} C_VEL
LIN {X 0,Y 435.156,Z 330.297,A -85,B 0,C 180,E1 -9465.215,E2 -9465.215} C_VEL
LIN {X 0,Y 435.391,Z 324.231,A -85,B 0,C 180,E1 -9465.566,E2 -9465.566} C_VEL
LIN {X 0,Y 433.586,Z 311.283,A -85,B 0,C 180,E1 -9466.209,E2 -9466.209} C_VEL
LIN {X 0,Y 431.438,Z 300.053,A -85,B 0,C 180,E1 -9466.635,E2 -9466.635} C_VEL
LIN {X 0,Y 431.343,Z 298.961,A -85,B 0,C 180,E1 -9466.67,E2 -9466.67} C_VEL
LIN {X 0,Y 431.468,Z 293.192,A -85,B 0,C 180,E1 -9470.002,E2 -9470.002} C_VEL
LIN {X 0,Y 431.65,Z 288.165,A -85,B 0,C 180,E1 -9473.001,E2 -9473.001} C_VEL
LIN {X 0,Y 431.855,Z 283.182,A -85,B 0,C 180,E1 -9476.065,E2 -9476.065} C_VEL
LIN {X 0,Y 432.101,Z 278.255,A -85,B 0,C 180,E1 -9479.205,E2 -9479.205} C_VEL
LIN {X 0,Y 432.481,Z 273.399,A -85,B 0,C 180,E1 -9482.429,E2 -9482.429} C_VEL
LIN {X 0,Y 432.79,Z 268.617,A -85,B 0,C 180,E1 -9485.774,E2 -9485.774} C_VEL
LIN {X 0,Y 433.099,Z 263.943,A -85,B 0,C 180,E1 -9489.26,E2 -9489.26} C_VEL
LIN {X 0,Y 433.278,Z 260.808,A -85,B 0,C 180,E1 -9491.738,E2 -9491.738} C_VEL
LIN {X 0,Y 433.092,Z 257.664,A -85,B 0,C 180,E1 -9494.434,E2 -9494.434} C_VEL
LIN {X 0,Y 432.747,Z 254.923,A -85,B 0,C 180,E1 -9496.988,E2 -9496.988} C_VEL
LIN {X 0,Y 432.317,Z 252.136,A -85,B 0,C 180,E1 -9499.822,E2 -9499.822} C_VEL
LIN {X 0,Y 432.31,Z 252.136,A -85,B 0,C 180,E1 -9503.018,E2 -9503.018} C_VEL
LIN {X 0,Y 432.339,Z 252.135,A -85,B 0,C 180,E1 -9505.998,E2 -9505.998} C_VEL
LIN {X 0,Y 432.351,Z 252.127,A -85,B 0,C 180,E1 -9509.486,E2 -9509.486} C_VEL
LIN {X 0,Y 432.34,Z 252.134,A -85,B 0,C 180,E1 -9511.869,E2 -9511.869} C_VEL
LIN {X 0,Y 432.38,Z 252.125,A -85,B 0,C 180,E1 -9515.535,E2 -9515.535} C_VEL
LIN {X 0,Y 432.351,Z 252.126,A -85,B 0,C 180,E1 -9519.042,E2 -9519.042} C_VEL
LIN {X 0,Y 432.359,Z 252.128,A -85,B 0,C 180,E1 -9522.006,E2 -9522.006} C_VEL
LIN {X 0,Y 432.393,Z 252.121,A -85,B 0,C 180,E1 -9524.922,E2 -9524.922} C_VEL
LIN {X 0,Y 432.456,Z 252.117,A -85,B 0,C 180,E1 -9527.799,E2 -9527.799} C_VEL
LIN {X 0,Y 432.457,Z 252.118,A -85,B 0,C 180,E1 -9531.585,E2 -9531.585} C_VEL
LIN {X 0,Y 432.578,Z 252.097,A -85,B 0,C 180,E1 -9534.401,E2 -9534.401} C_VEL
LIN {X 0,Y 432.587,Z 252.096,A -85,B 0,C 180,E1 -9538.133,E2 -9538.133} C_VEL
LIN {X 0,Y 432.717,Z 252.08,A -85,B 0,C 180,E1 -9539.995,E2 -9539.995} C_VEL
LIN {X 0,Y 432.576,Z 252.1,A -85,B 0,C 180,E1 -9542.788,E2 -9542.788} C_VEL
LIN {X 0,Y 432.534,Z 252.104,A -85,B 0,C 180,E1 -9546.525,E2 -9546.525} C_VEL
LIN {X 0,Y 432.421,Z 252.12,A -85,B 0,C 180,E1 -9549.347,E2 -9549.347} C_VEL
LIN {X 0,Y 432.411,Z 252.124,A -85,B 0,C 180,E1 -9552.797,E2 -9552.797} C_VEL
LIN {X 0,Y 432.388,Z 252.124,A -85,B 0,C 180,E1 -9556.472,E2 -9556.472} C_VEL
LIN {X 0,Y 432.312,Z 252.131,A -85,B 0,C 180,E1 -9559.955,E2 -9559.955} C_VEL
LIN {X 0,Y 432.289,Z 252.137,A -85,B 0,C 180,E1 -9562.958,E2 -9562.958} C_VEL
LIN {X 0,Y 432.33,Z 252.129,A -85,B 0,C 180,E1 -9566.027,E2 -9566.027} C_VEL
LIN {X 0,Y 432.308,Z 252.132,A -85,B 0,C 180,E1 -9569.182,E2 -9569.182} C_VEL
LIN {X 0,Y 432.285,Z 252.141,A -85,B 0,C 180,E1 -9572.437,E2 -9572.437} C_VEL
LIN {X 0,Y 432.305,Z 252.132,A -85,B 0,C 180,E1 -9575.627,E2 -9575.627} C_VEL
LIN {X 0,Y 432.315,Z 252.132,A -85,B 0,C 180,E1 -9578.712,E2 -9578.712} C_VEL
LIN {X 0,Y 432.33,Z 252.131,A -85,B 0,C 180,E1 -9581.787,E2 -9581.787} C_VEL
LIN {X 0,Y 432.36,Z 252.129,A -85,B 0,C 180,E1 -9584.34,E2 -9584.34} C_VEL
LIN {X 0,Y 432.317,Z 252.13,A -85,B 0,C 180,E1 -9587.004,E2 -9587.004} C_VEL
LIN {X 0,Y 432.309,Z 252.136,A -85,B 0,C 180,E1 -9589.812,E2 -9589.812} C_VEL
LIN {X 0,Y 432.263,Z 252.136,A -85,B 0,C 180,E1 -9593.019,E2 -9593.019} C_VEL
LIN {X 0,Y 432.304,Z 252.137,A -85,B 0,C 180,E1 -9595.993,E2 -9595.993} C_VEL
LIN {X 0,Y 432.336,Z 252.135,A -85,B 0,C 180,E1 -9599.74,E2 -9599.74} C_VEL
LIN {X 0,Y 432.34,Z 252.131,A -85,B 0,C 180,E1 -9603.369,E2 -9603.369} C_VEL
LIN {X 0,Y 432.32,Z 252.132,A -85,B 0,C 180,E1 -9606.021,E2 -9606.021} C_VEL
LIN {X 0,Y 432.315,Z 252.132,A -85,B 0,C 180,E1 -9609.045,E2 -9609.045} C_VEL
LIN {X 0,Y 432.32,Z 252.134,A -85,B 0,C 180,E1 -9612.009,E2 -9612.009} C_VEL
LIN {X 0,Y 432.348,Z 252.132,A -85,B 0,C 180,E1 -9614.925,E2 -9614.925} C_VEL
LIN {X 0,Y 432.419,Z 252.12,A -85,B 0,C 180,E1 -9617.803,E2 -9617.803} C_VEL
LIN {X 0,Y 432.432,Z 252.12,A -85,B 0,C 180,E1 -9621.589,E2 -9621.589} C_VEL
LIN {X 0,Y 432.542,Z 252.105,A -85,B 0,C 180,E1 -9624.406,E2 -9624.406} C_VEL
LIN {X 0,Y 432.541,Z 252.105,A -85,B 0,C 180,E1 -9628.138,E2 -9628.138} C_VEL
LIN {X 0,Y 432.668,Z 252.091,A -85,B 0,C 180,E1 -9630,E2 -9630} C_VEL
LIN {X 0,Y 432.548,Z 252.107,A -85,B 0,C 180,E1 -9632.794,E2 -9632.794} C_VEL
LIN {X 0,Y 432.404,Z 252.122,A -85,B 0,C 180,E1 -9635.004,E2 -9635.004} C_VEL
LIN {X 0,Y 431.846,Z 252.192,A -85,B 0,C 180,E1 -9635.782,E2 -9635.782} C_VEL
LIN {X 0,Y 429.012,Z 252.547,A -85,B 0,C 180,E1 -9637.047,E2 -9637.047} C_VEL
LIN {X 0,Y 426.534,Z 252.855,A -85,B 0,C 180,E1 -9638.069,E2 -9638.069} C_VEL
LIN {X 0,Y 425.45,Z 252.992,A -85,B 0,C 180,E1 -9638.858,E2 -9638.858} C_VEL
LIN {X 0,Y 425.355,Z 253.001,A -85,B 0,C 180,E1 -9639.126,E2 -9639.126} C_VEL
LIN {X 0,Y 425.34,Z 253.005,A -85,B 0,C 180,E1 -9642.912,E2 -9642.912} C_VEL
LIN {X 0,Y 425.307,Z 253.01,A -85,B 0,C 180,E1 -9646.611,E2 -9646.611} C_VEL
LIN {X 0,Y 425.3,Z 253.006,A -85,B 0,C 180,E1 -9649.651,E2 -9649.651} C_VEL
LIN {X 0,Y 425.276,Z 253.013,A -85,B 0,C 180,E1 -9652.339,E2 -9652.339} C_VEL
LIN {X 0,Y 425.241,Z 253.011,A -85,B 0,C 180,E1 -9655.448,E2 -9655.448} C_VEL
LIN {X 0,Y 425.279,Z 253.01,A -85,B 0,C 180,E1 -9658.635,E2 -9658.635} C_VEL
LIN {X 0,Y 425.209,Z 253.019,A -85,B 0,C 180,E1 -9661.931,E2 -9661.931} C_VEL
LIN {X 0,Y 425.245,Z 253.011,A -85,B 0,C 180,E1 -9665.34,E2 -9665.34} C_VEL
LIN {X 0,Y 425.264,Z 253.008,A -85,B 0,C 180,E1 -9669.051,E2 -9669.051} C_VEL
LIN {X 0,Y 425.282,Z 253.007,A -85,B 0,C 180,E1 -9672.651,E2 -9672.651} C_VEL
LIN {X 0,Y 425.308,Z 253.007,A -85,B 0,C 180,E1 -9676.061,E2 -9676.061} C_VEL
LIN {X 0,Y 425.265,Z 253.008,A -85,B 0,C 180,E1 -9678.631,E2 -9678.631} C_VEL
LIN {X 0,Y 425.279,Z 253.007,A -85,B 0,C 180,E1 -9681.109,E2 -9681.109} C_VEL
LIN {X 0,Y 425.261,Z 253.009,A -85,B 0,C 180,E1 -9684.67,E2 -9684.67} C_VEL
LIN {X 0,Y 425.227,Z 253.014,A -85,B 0,C 180,E1 -9688.079,E2 -9688.079} C_VEL
LIN {X 0,Y 425.297,Z 253.01,A -85,B 0,C 180,E1 -9691.374,E2 -9691.374} C_VEL
LIN {X 0,Y 425.261,Z 253.009,A -85,B 0,C 180,E1 -9694.56,E2 -9694.56} C_VEL
LIN {X 0,Y 425.26,Z 253.012,A -85,B 0,C 180,E1 -9697.667,E2 -9697.667} C_VEL
LIN {X 0,Y 425.335,Z 253.001,A -85,B 0,C 180,E1 -9700.71,E2 -9700.71} C_VEL
LIN {X 0,Y 425.365,Z 252.997,A -85,B 0,C 180,E1 -9703.694,E2 -9703.694} C_VEL
LIN {X 0,Y 425.392,Z 252.994,A -85,B 0,C 180,E1 -9707.604,E2 -9707.604} C_VEL
LIN {X 0,Y 425.391,Z 252.994,A -85,B 0,C 180,E1 -9711.455,E2 -9711.455} C_VEL
LIN {X 0,Y 425.527,Z 252.977,A -85,B 0,C 180,E1 -9714.319,E2 -9714.319} C_VEL
LIN {X 0,Y 425.561,Z 252.972,A -85,B 0,C 180,E1 -9718.113,E2 -9718.113} C_VEL
LIN {X 0,Y 425.687,Z 252.956,A -85,B 0,C 180,E1 -9720.006,E2 -9720.006} C_VEL
LIN {X 0,Y 425.512,Z 252.983,A -85,B 0,C 180,E1 -9722.846,E2 -9722.846} C_VEL
LIN {X 0,Y 425.534,Z 252.975,A -85,B 0,C 180,E1 -9725.692,E2 -9725.692} C_VEL
LIN {X 0,Y 425.402,Z 252.999,A -85,B 0,C 180,E1 -9728.556,E2 -9728.556} C_VEL
LIN {X 0,Y 425.409,Z 252.997,A -85,B 0,C 180,E1 -9732.407,E2 -9732.407} C_VEL
LIN {X 0,Y 425.387,Z 253,A -85,B 0,C 180,E1 -9736.317,E2 -9736.317} C_VEL
LIN {X 0,Y 425.33,Z 253.001,A -85,B 0,C 180,E1 -9739.64,E2 -9739.64} C_VEL
LIN {X 0,Y 425.291,Z 253.011,A -85,B 0,C 180,E1 -9742.343,E2 -9742.343} C_VEL
LIN {X 0,Y 425.322,Z 253.003,A -85,B 0,C 180,E1 -9744.661,E2 -9744.661} C_VEL
LIN {X 0,Y 425.263,Z 253.01,A -85,B 0,C 180,E1 -9747.568,E2 -9747.568} C_VEL
LIN {X 0,Y 425.296,Z 253.005,A -85,B 0,C 180,E1 -9750.765,E2 -9750.765} C_VEL
LIN {X 0,Y 425.306,Z 253.009,A -85,B 0,C 180,E1 -9754.289,E2 -9754.289} C_VEL
LIN {X 0,Y 425.282,Z 253.013,A -85,B 0,C 180,E1 -9757.698,E2 -9757.698} C_VEL
LIN {X 0,Y 425.307,Z 253.239,A -85,B 0,C 180,E1 -9760.129,E2 -9760.129} C_VEL
LIN {X 0,Y 425.776,Z 256.501,A -85,B 0,C 180,E1 -9763.426,E2 -9763.426} C_VEL
LIN {X 0,Y 426.136,Z 259.445,A -85,B 0,C 180,E1 -9766.159,E2 -9766.159} C_VEL
LIN {X 0,Y 426.204,Z 262.446,A -85,B 0,C 180,E1 -9768.733,E2 -9768.733} C_VEL
LIN {X 0,Y 426.036,Z 265.501,A -85,B 0,C 180,E1 -9771.182,E2 -9771.182} C_VEL
LIN {X 0,Y 425.691,Z 270.214,A -85,B 0,C 180,E1 -9774.702,E2 -9774.702} C_VEL
LIN {X 0,Y 425.347,Z 274.97,A -85,B 0,C 180,E1 -9778.081,E2 -9778.081} C_VEL
LIN {X 0,Y 424.993,Z 279.824,A -85,B 0,C 180,E1 -9781.344,E2 -9781.344} C_VEL
LIN {X 0,Y 424.717,Z 284.75,A -85,B 0,C 180,E1 -9784.518,E2 -9784.518} C_VEL
LIN {X 0,Y 424.507,Z 289.723,A -85,B 0,C 180,E1 -9787.619,E2 -9787.619} C_VEL
LIN {X 0,Y 424.351,Z 294.882,A -85,B 0,C 180,E1 -9790.745,E2 -9790.745} C_VEL
LIN {X 0,Y 424.264,Z 298.781,A -85,B 0,C 180,E1 -9793.048,E2 -9793.048} C_VEL
LIN {X 0,Y 426.276,Z 309.513,A -85,B 0,C 180,E1 -9793.45,E2 -9793.45} C_VEL
LIN {X 0,Y 427.913,Z 320.431,A -85,B 0,C 180,E1 -9793.979,E2 -9793.979} C_VEL
LIN {X 0,Y 428.473,Z 326.147,A -85,B 0,C 180,E1 -9794.303,E2 -9794.303} C_VEL
LIN {X 0,Y 427.968,Z 335.589,A -85,B 0,C 180,E1 -9794.889,E2 -9794.889} C_VEL
LIN {X 0,Y 427.365,Z 344.866,A -85,B 0,C 180,E1 -9795.598,E2 -9795.598} C_VEL
LIN {X 0,Y 426.802,Z 353.692,A -85,B 0,C 180,E1 -9796.416,E2 -9796.416} C_VEL
LIN {X 0,Y 426.268,Z 362.346,A -85,B 0,C 180,E1 -9797.382,E2 -9797.382} C_VEL
LIN {X 0,Y 425.781,Z 369.566,A -85,B 0,C 180,E1 -9798.335,E2 -9798.335} C_VEL
LIN {X 0,Y 425.31,Z 375.767,A -85,B 0,C 180,E1 -9799.287,E2 -9799.287} C_VEL
LIN {X 0,Y 424.883,Z 382.305,A -85,B 0,C 180,E1 -9800.479,E2 -9800.479} C_VEL
LIN {X 0,Y 424.645,Z 386.807,A -85,B 0,C 180,E1 -9801.434,E2 -9801.434} C_VEL
LIN {X 0,Y 424.365,Z 392.298,A -85,B 0,C 180,E1 -9802.865,E2 -9802.865} C_VEL
LIN {X 0,Y 424.199,Z 396.621,A -85,B 0,C 180,E1 -9804.295,E2 -9804.295} C_VEL
LIN {X 0,Y 424.206,Z 398.988,A -85,B 0,C 180,E1 -9805.248,E2 -9805.248} C_VEL
LIN {X 0,Y 424.088,Z 400.783,A -85,B 0,C 180,E1 -9806.199,E2 -9806.199} C_VEL
LIN {X 0,Y 424.134,Z 403.228,A -85,B 0,C 180,E1 -9808.101,E2 -9808.101} C_VEL
LIN {X 0,Y 424.075,Z 403.814,A -85,B 0,C 180,E1 -9809.05,E2 -9809.05} C_VEL
LIN {X 0,Y 424.075,Z 403.814,A -85,B 0,C 180,E1 -9810.95,E2 -9810.95} C_VEL
LIN {X 0,Y 424.134,Z 403.228,A -85,B 0,C 180,E1 -9811.899,E2 -9811.899} C_VEL
LIN {X 0,Y 424.088,Z 400.783,A -85,B 0,C 180,E1 -9813.801,E2 -9813.801} C_VEL
LIN {X 0,Y 424.212,Z 397.839,A -85,B 0,C 180,E1 -9815.228,E2 -9815.228} C_VEL
LIN {X 0,Y 424.313,Z 393.852,A -85,B 0,C 180,E1 -9816.658,E2 -9816.658} C_VEL
LIN {X 0,Y 424.535,Z 388.723,A -85,B 0,C 180,E1 -9818.089,E2 -9818.089} C_VEL
LIN {X 0,Y 424.811,Z 383.461,A -85,B 0,C 180,E1 -9819.282,E2 -9819.282} C_VEL
LIN {X 0,Y 425.216,Z 377.144,A -85,B 0,C 180,E1 -9820.475,E2 -9820.475} C_VEL
LIN {X 0,Y 425.642,Z 371.193,A -85,B 0,C 180,E1 -9821.428,E2 -9821.428} C_VEL
LIN {X 0,Y 426.154,Z 364.266,A -85,B 0,C 180,E1 -9822.38,E2 -9822.38} C_VEL
LIN {X 0,Y 426.663,Z 356.083,A -85,B 0,C 180,E1 -9823.333,E2 -9823.333} C_VEL
LIN {X 0,Y 427.158,Z 347.319,A -85,B 0,C 180,E1 -9824.188,E2 -9824.188} C_VEL
LIN {X 0,Y 427.727,Z 338.852,A -85,B 0,C 180,E1 -9824.876,E2 -9824.876} C_VEL
LIN {X 0,Y 428.32,Z 330.139,A -85,B 0,C 180,E1 -9825.461,E2 -9825.461} C_VEL
LIN {X 0,Y 428.381,Z 324.13,A -85,B 0,C 180,E1 -9825.822,E2 -9825.822} C_VEL
LIN {X 0,Y 426.503,Z 310.904,A -85,B 0,C 180,E1 -9826.492,E2 -9826.492} C_VEL
LIN {X 0,Y 424.405,Z 299.991,A -85,B 0,C 180,E1 -9826.916,E2 -9826.916} C_VEL
LIN {X 0,Y 424.262,Z 298.781,A -85,B 0,C 180,E1 -9826.953,E2 -9826.953} C_VEL
LIN {X 0,Y 424.398,Z 293.053,A -85,B 0,C 180,E1 -9830.35,E2 -9830.35} C_VEL
LIN {X 0,Y 424.582,Z 288.051,A -85,B 0,C 180,E1 -9833.407,E2 -9833.407} C_VEL
LIN {X 0,Y 424.821,Z 282.833,A -85,B 0,C 180,E1 -9836.698,E2 -9836.698} C_VEL
LIN {X 0,Y 425.099,Z 278.193,A -85,B 0,C 180,E1 -9839.733,E2 -9839.733} C_VEL
LIN {X 0,Y 425.477,Z 273.355,A -85,B 0,C 180,E1 -9843.03,E2 -9843.03} C_VEL
LIN {X 0,Y 425.769,Z 269.195,A -85,B 0,C 180,E1 -9846.014,E2 -9846.014} C_VEL
LIN {X 0,Y 426.071,Z 265.048,A -85,B 0,C 180,E1 -9849.167,E2 -9849.167} C_VEL
LIN {X 0,Y 426.238,Z 261.423,A -85,B 0,C 180,E1 -9852.095,E2 -9852.095} C_VEL
LIN {X 0,Y 426.034,Z 258.349,A -85,B 0,C 180,E1 -9854.814,E2 -9854.814} C_VEL
LIN {X 0,Y 425.567,Z 255.046,A -85,B 0,C 180,E1 -9857.999,E2 -9857.999} C_VEL
LIN {X 0,Y 425.307,Z 253.24,A -85,B 0,C 180,E1 -9859.871,E2 -9859.871} C_VEL
LIN {X 0,Y 425.282,Z 253.013,A -85,B 0,C 180,E1 -9862.486,E2 -9862.486} C_VEL
LIN {X 0,Y 425.292,Z 253.013,A -85,B 0,C 180,E1 -9865.812,E2 -9865.812} C_VEL
LIN {X 0,Y 425.296,Z 253.005,A -85,B 0,C 180,E1 -9869.235,E2 -9869.235} C_VEL
LIN {X 0,Y 425.263,Z 253.01,A -85,B 0,C 180,E1 -9872.432,E2 -9872.432} C_VEL
LIN {X 0,Y 425.349,Z 253.002,A -85,B 0,C 180,E1 -9875.598,E2 -9875.598} C_VEL
LIN {X 0,Y 425.294,Z 253.004,A -85,B 0,C 180,E1 -9878.677,E2 -9878.677} C_VEL
LIN {X 0,Y 425.321,Z 253.009,A -85,B 0,C 180,E1 -9881.698,E2 -9881.698} C_VEL
LIN {X 0,Y 425.346,Z 252.998,A -85,B 0,C 180,E1 -9884.666,E2 -9884.666} C_VEL
LIN {X 0,Y 425.409,Z 252.997,A -85,B 0,C 180,E1 -9887.593,E2 -9887.593} C_VEL
LIN {X 0,Y 425.402,Z 252.999,A -85,B 0,C 180,E1 -9891.444,E2 -9891.444} C_VEL
LIN {X 0,Y 425.534,Z 252.975,A -85,B 0,C 180,E1 -9894.308,E2 -9894.308} C_VEL
LIN {X 0,Y 425.556,Z 252.972,A -85,B 0,C 180,E1 -9898.102,E2 -9898.102} C_VEL
LIN {X 0,Y 425.687,Z 252.956,A -85,B 0,C 180,E1 -9899.994,E2 -9899.994} C_VEL
LIN {X 0,Y 425.53,Z 252.978,A -85,B 0,C 180,E1 -9902.834,E2 -9902.834} C_VEL
LIN {X 0,Y 425.489,Z 252.982,A -85,B 0,C 180,E1 -9906.603,E2 -9906.603} C_VEL
LIN {X 0,Y 425.38,Z 252.996,A -85,B 0,C 180,E1 -9909.504,E2 -9909.504} C_VEL
LIN {X 0,Y 425.373,Z 253.002,A -85,B 0,C 180,E1 -9912.898,E2 -9912.898} C_VEL
LIN {X 0,Y 425.337,Z 253.004,A -85,B 0,C 180,E1 -9916.598,E2 -9916.598} C_VEL
LIN {X 0,Y 425.302,Z 253.003,A -85,B 0,C 180,E1 -9919.629,E2 -9919.629} C_VEL
LIN {X 0,Y 425.26,Z 253.012,A -85,B 0,C 180,E1 -9922.333,E2 -9922.333} C_VEL
LIN {X 0,Y 425.261,Z 253.009,A -85,B 0,C 180,E1 -9925.44,E2 -9925.44} C_VEL
LIN {X 0,Y 425.297,Z 253.01,A -85,B 0,C 180,E1 -9928.626,E2 -9928.626} C_VEL
LIN {X 0,Y 425.227,Z 253.014,A -85,B 0,C 180,E1 -9931.921,E2 -9931.921} C_VEL
LIN {X 0,Y 425.261,Z 253.009,A -85,B 0,C 180,E1 -9935.33,E2 -9935.33} C_VEL
LIN {X 0,Y 425.267,Z 253.008,A -85,B 0,C 180,E1 -9939.04,E2 -9939.04} C_VEL
LIN {X 0,Y 425.291,Z 253.007,A -85,B 0,C 180,E1 -9942.64,E2 -9942.64} C_VEL
LIN {X 0,Y 425.287,Z 253.012,A -85,B 0,C 180,E1 -9946.049,E2 -9946.049} C_VEL
LIN {X 0,Y 425.26,Z 253.01,A -85,B 0,C 180,E1 -9948.621,E2 -9948.621} C_VEL
LIN {X 0,Y 425.274,Z 253.007,A -85,B 0,C 180,E1 -9951.1,E2 -9951.1} C_VEL
LIN {X 0,Y 425.245,Z 253.011,A -85,B 0,C 180,E1 -9954.66,E2 -9954.66} C_VEL
LIN {X 0,Y 425.209,Z 253.019,A -85,B 0,C 180,E1 -9958.069,E2 -9958.069} C_VEL
LIN {X 0,Y 425.279,Z 253.01,A -85,B 0,C 180,E1 -9961.365,E2 -9961.365} C_VEL
LIN {X 0,Y 425.241,Z 253.011,A -85,B 0,C 180,E1 -9964.552,E2 -9964.552} C_VEL
LIN {X 0,Y 425.268,Z 253.013,A -85,B 0,C 180,E1 -9967.714,E2 -9967.714} C_VEL
LIN {X 0,Y 425.303,Z 253.004,A -85,B 0,C 180,E1 -9970.702,E2 -9970.702} C_VEL
LIN {X 0,Y 425.336,Z 253.005,A -85,B 0,C 180,E1 -9973.687,E2 -9973.687} C_VEL
LIN {X 0,Y 425.367,Z 253,A -85,B 0,C 180,E1 -9977.597,E2 -9977.597} C_VEL
LIN {X 0,Y 425.401,Z 252.997,A -85,B 0,C 180,E1 -9981.449,E2 -9981.449} C_VEL
LIN {X 0,Y 425.52,Z 252.98,A -85,B 0,C 180,E1 -9984.313,E2 -9984.313} C_VEL
LIN {X 0,Y 425.51,Z 252.981,A -85,B 0,C 180,E1 -9988.107,E2 -9988.107} C_VEL
LIN {X 0,Y 425.638,Z 252.967,A -85,B 0,C 180,E1 -9990,E2 -9990} C_VEL
LIN {X 0,Y 425.5,Z 252.985,A -85,B 0,C 180,E1 -9992.84,E2 -9992.84} C_VEL
LIN {X 0,Y 425.52,Z 252.98,A -85,B 0,C 180,E1 -9995.687,E2 -9995.687} C_VEL
LIN {X 0,Y 425.401,Z 252.997,A -85,B 0,C 180,E1 -9998.551,E2 -9998.551} C_VEL
LIN {X 0,Y 425.355,Z 253.001,A -85,B 0,C 180,E1 -9999.126,E2 -9999.126} C_VEL
LIN {X 0,Y 424.674,Z 253.087,A -85,B 0,C 180,E1 -9999.916,E2 -9999.916} C_VEL
LIN {X 0,Y 421.822,Z 253.445,A -85,B 0,C 180,E1 -10001.2,E2 -10001.2} C_VEL
LIN {X 0,Y 419.41,Z 253.745,A -85,B 0,C 180,E1 -10002.236,E2 -10002.236} C_VEL
LIN {X 0,Y 418.364,Z 253.874,A -85,B 0,C 180,E1 -10003.037,E2 -10003.037} C_VEL
LIN {X 0,Y 418.272,Z 253.884,A -85,B 0,C 180,E1 -10003.309,E2 -10003.309} C_VEL
LIN {X 0,Y 418.257,Z 253.888,A -85,B 0,C 180,E1 -10006.741,E2 -10006.741} C_VEL
LIN {X 0,Y 418.242,Z 253.887,A -85,B 0,C 180,E1 -10009.805,E2 -10009.805} C_VEL
LIN {X 0,Y 418.229,Z 253.888,A -85,B 0,C 180,E1 -10012.736,E2 -10012.736} C_VEL
LIN {X 0,Y 418.214,Z 253.889,A -85,B 0,C 180,E1 -10015.907,E2 -10015.907} C_VEL
LIN {X 0,Y 418.216,Z 253.886,A -85,B 0,C 180,E1 -10019.165,E2 -10019.165} C_VEL
LIN {X 0,Y 418.201,Z 253.889,A -85,B 0,C 180,E1 -10022.848,E2 -10022.848} C_VEL
LIN {X 0,Y 418.195,Z 253.894,A -85,B 0,C 180,E1 -10026.243,E2 -10026.243} C_VEL
LIN {X 0,Y 418.217,Z 253.889,A -85,B 0,C 180,E1 -10029.685,E2 -10029.685} C_VEL
LIN {X 0,Y 418.236,Z 253.887,A -85,B 0,C 180,E1 -10032.334,E2 -10032.334} C_VEL
LIN {X 0,Y 418.239,Z 253.884,A -85,B 0,C 180,E1 -10035.121,E2 -10035.121} C_VEL
LIN {X 0,Y 418.25,Z 253.889,A -85,B 0,C 180,E1 -10037.779,E2 -10037.779} C_VEL
LIN {X 0,Y 418.222,Z 253.891,A -85,B 0,C 180,E1 -10041.565,E2 -10041.565} C_VEL
LIN {X 0,Y 418.221,Z 253.888,A -85,B 0,C 180,E1 -10045.165,E2 -10045.165} C_VEL
LIN {X 0,Y 418.208,Z 253.893,A -85,B 0,C 180,E1 -10047.478,E2 -10047.478} C_VEL
LIN {X 0,Y 418.235,Z 253.885,A -85,B 0,C 180,E1 -10050.901,E2 -10050.901} C_VEL
LIN {X 0,Y 418.237,Z 253.884,A -85,B 0,C 180,E1 -10054.102,E2 -10054.102} C_VEL
LIN {X 0,Y 418.204,Z 253.894,A -85,B 0,C 180,E1 -10057.269,E2 -10057.269} C_VEL
LIN {X 0,Y 418.257,Z 253.881,A -85,B 0,C 180,E1 -10060.37,E2 -10060.37} C_VEL
LIN {X 0,Y 418.293,Z 253.881,A -85,B 0,C 180,E1 -10063.411,E2 -10063.411} C_VEL
LIN {X 0,Y 418.326,Z 253.879,A -85,B 0,C 180,E1 -10067.006,E2 -10067.006} C_VEL
LIN {X 0,Y 418.321,Z 253.874,A -85,B 0,C 180,E1 -10070.334,E2 -10070.334} C_VEL
LIN {X 0,Y 418.452,Z 253.86,A -85,B 0,C 180,E1 -10073.254,E2 -10073.254} C_VEL
LIN {X 0,Y 418.317,Z 253.877,A -85,B 0,C 180,E1 -10075.187,E2 -10075.187} C_VEL
LIN {X 0,Y 418.53,Z 253.848,A -85,B 0,C 180,E1 -10078.081,E2 -10078.081} C_VEL
LIN {X 0,Y 418.656,Z 253.832,A -85,B 0,C 180,E1 -10080.006,E2 -10080.006} C_VEL
LIN {X 0,Y 418.469,Z 253.859,A -85,B 0,C 180,E1 -10082.893,E2 -10082.893} C_VEL
LIN {X 0,Y 418.493,Z 253.852,A -85,B 0,C 180,E1 -10085.788,E2 -10085.788} C_VEL
LIN {X 0,Y 418.372,Z 253.872,A -85,B 0,C 180,E1 -10088.701,E2 -10088.701} C_VEL
LIN {X 0,Y 418.31,Z 253.875,A -85,B 0,C 180,E1 -10091.636,E2 -10091.636} C_VEL
LIN {X 0,Y 418.3,Z 253.881,A -85,B 0,C 180,E1 -10094.602,E2 -10094.602} C_VEL
LIN {X 0,Y 418.279,Z 253.879,A -85,B 0,C 180,E1 -10097.609,E2 -10097.609} C_VEL
LIN {X 0,Y 418.251,Z 253.884,A -85,B 0,C 180,E1 -10100.668,E2 -10100.668} C_VEL
LIN {X 0,Y 418.276,Z 253.882,A -85,B 0,C 180,E1 -10103.786,E2 -10103.786} C_VEL
LIN {X 0,Y 418.219,Z 253.886,A -85,B 0,C 180,E1 -10107.049,E2 -10107.049} C_VEL
LIN {X 0,Y 418.247,Z 253.886,A -85,B 0,C 180,E1 -10110.276,E2 -10110.276} C_VEL
LIN {X 0,Y 418.244,Z 253.887,A -85,B 0,C 180,E1 -10113.682,E2 -10113.682} C_VEL
LIN {X 0,Y 418.245,Z 253.888,A -85,B 0,C 180,E1 -10117.228,E2 -10117.228} C_VEL
LIN {X 0,Y 418.253,Z 253.997,A -85,B 0,C 180,E1 -10119.686,E2 -10119.686} C_VEL
LIN {X 0,Y 418.646,Z 256.56,A -85,B 0,C 180,E1 -10122.385,E2 -10122.385} C_VEL
LIN {X 0,Y 419.02,Z 259.479,A -85,B 0,C 180,E1 -10125.217,E2 -10125.217} C_VEL
LIN {X 0,Y 419.226,Z 262.467,A -85,B 0,C 180,E1 -10127.89,E2 -10127.89} C_VEL
LIN {X 0,Y 419.048,Z 265.625,A -85,B 0,C 180,E1 -10130.492,E2 -10130.492} C_VEL
LIN {X 0,Y 418.757,Z 269.706,A -85,B 0,C 180,E1 -10133.671,E2 -10133.671} C_VEL
LIN {X 0,Y 418.419,Z 274.425,A -85,B 0,C 180,E1 -10137.127,E2 -10137.127} C_VEL
LIN {X 0,Y 418.096,Z 278.13,A -85,B 0,C 180,E1 -10139.717,E2 -10139.717} C_VEL
LIN {X 0,Y 417.774,Z 283.153,A -85,B 0,C 180,E1 -10143.079,E2 -10143.079} C_VEL
LIN {X 0,Y 417.533,Z 287.94,A -85,B 0,C 180,E1 -10146.174,E2 -10146.174} C_VEL
LIN {X 0,Y 417.349,Z 292.917,A -85,B 0,C 180,E1 -10149.291,E2 -10149.291} C_VEL
LIN {X 0,Y 417.154,Z 298.585,A -85,B 0,C 180,E1 -10152.745,E2 -10152.745} C_VEL
LIN {X 0,Y 419.513,Z 310.976,A -85,B 0,C 180,E1 -10153.235,E2 -10153.235} C_VEL
LIN {X 0,Y 421.433,Z 324.614,A -85,B 0,C 180,E1 -10153.951,E2 -10153.951} C_VEL
LIN {X 0,Y 421.405,Z 330.21,A -85,B 0,C 180,E1 -10154.295,E2 -10154.295} C_VEL
LIN {X 0,Y 420.676,Z 341.9,A -85,B 0,C 180,E1 -10155.116,E2 -10155.116} C_VEL
LIN {X 0,Y 419.915,Z 352.789,A -85,B 0,C 180,E1 -10156.112,E2 -10156.112} C_VEL
LIN {X 0,Y 419.447,Z 360.23,A -85,B 0,C 180,E1 -10156.927,E2 -10156.927} C_VEL
LIN {X 0,Y 418.803,Z 369.371,A -85,B 0,C 180,E1 -10158.137,E2 -10158.137} C_VEL
LIN {X 0,Y 418.308,Z 375.572,A -85,B 0,C 180,E1 -10159.105,E2 -10159.105} C_VEL
LIN {X 0,Y 417.848,Z 382.109,A -85,B 0,C 180,E1 -10160.317,E2 -10160.317} C_VEL
LIN {X 0,Y 417.582,Z 386.611,A -85,B 0,C 180,E1 -10161.288,E2 -10161.288} C_VEL
LIN {X 0,Y 417.293,Z 392.103,A -85,B 0,C 180,E1 -10162.744,E2 -10162.744} C_VEL
LIN {X 0,Y 417.117,Z 396.426,A -85,B 0,C 180,E1 -10164.198,E2 -10164.198} C_VEL
LIN {X 0,Y 417.114,Z 398.793,A -85,B 0,C 180,E1 -10165.167,E2 -10165.167} C_VEL
LIN {X 0,Y 417.025,Z 401.976,A -85,B 0,C 180,E1 -10167.102,E2 -10167.102} C_VEL
LIN {X 0,Y 417.061,Z 403.034,A -85,B 0,C 180,E1 -10168.069,E2 -10168.069} C_VEL
LIN {X 0,Y 416.999,Z 403.62,A -85,B 0,C 180,E1 -10169.034,E2 -10169.034} C_VEL
LIN {X 0,Y 416.999,Z 403.62,A -85,B 0,C 180,E1 -10170.966,E2 -10170.966} C_VEL
LIN {X 0,Y 417.061,Z 403.034,A -85,B 0,C 180,E1 -10171.931,E2 -10171.931} C_VEL
LIN {X 0,Y 417.005,Z 400.589,A -85,B 0,C 180,E1 -10173.865,E2 -10173.865} C_VEL
LIN {X 0,Y 417.128,Z 397.644,A -85,B 0,C 180,E1 -10175.317,E2 -10175.317} C_VEL
LIN {X 0,Y 417.247,Z 393.657,A -85,B 0,C 180,E1 -10176.771,E2 -10176.771} C_VEL
LIN {X 0,Y 417.474,Z 388.527,A -85,B 0,C 180,E1 -10178.227,E2 -10178.227} C_VEL
LIN {X 0,Y 417.778,Z 383.265,A -85,B 0,C 180,E1 -10179.44,E2 -10179.44} C_VEL
LIN {X 0,Y 418.189,Z 376.948,A -85,B 0,C 180,E1 -10180.653,E2 -10180.653} C_VEL
LIN {X 0,Y 418.647,Z 370.997,A -85,B 0,C 180,E1 -10181.621,E2 -10181.621} C_VEL
LIN {X 0,Y 419.182,Z 364.07,A -85,B 0,C 180,E1 -10182.589,E2 -10182.589} C_VEL
LIN {X 0,Y 419.744,Z 355.888,A -85,B 0,C 180,E1 -10183.556,E2 -10183.556} C_VEL
LIN {X 0,Y 420.248,Z 347.255,A -85,B 0,C 180,E1 -10184.415,E2 -10184.415} C_VEL
LIN {X 0,Y 420.841,Z 338.657,A -85,B 0,C 180,E1 -10185.125,E2 -10185.125} C_VEL
LIN {X 0,Y 421.442,Z 330.212,A -85,B 0,C 180,E1 -10185.704,E2 -10185.704} C_VEL
LIN {X 0,Y 421.463,Z 324.618,A -85,B 0,C 180,E1 -10186.047,E2 -10186.047} C_VEL
LIN {X 0,Y 419.559,Z 311.358,A -85,B 0,C 180,E1 -10186.75,E2 -10186.75} C_VEL
LIN {X 0,Y 417.375,Z 300.226,A -85,B 0,C 180,E1 -10187.2,E2 -10187.2} C_VEL
LIN {X 0,Y 417.137,Z 298.553,A -85,B 0,C 180,E1 -10187.274,E2 -10187.274} C_VEL
LIN {X 0,Y 417.348,Z 292.914,A -85,B 0,C 180,E1 -10190.709,E2 -10190.709} C_VEL
LIN {X 0,Y 417.536,Z 287.937,A -85,B 0,C 180,E1 -10193.826,E2 -10193.826} C_VEL
LIN {X 0,Y 417.779,Z 283.004,A -85,B 0,C 180,E1 -10197.013,E2 -10197.013} C_VEL
LIN {X 0,Y 418.101,Z 278.123,A -85,B 0,C 180,E1 -10200.283,E2 -10200.283} C_VEL
LIN {X 0,Y 418.421,Z 274.403,A -85,B 0,C 180,E1 -10202.874,E2 -10202.874} C_VEL
LIN {X 0,Y 418.756,Z 269.689,A -85,B 0,C 180,E1 -10206.329,E2 -10206.329} C_VEL
LIN {X 0,Y 419.054,Z 265.491,A -85,B 0,C 180,E1 -10209.59,E2 -10209.59} C_VEL
LIN {X 0,Y 419.206,Z 262.041,A -85,B 0,C 180,E1 -10212.463,E2 -10212.463} C_VEL
LIN {X 0,Y 418.974,Z 259.023,A -85,B 0,C 180,E1 -10215.205,E2 -10215.205} C_VEL
LIN {X 0,Y 418.582,Z 256.375,A -85,B 0,C 180,E1 -10217.805,E2 -10217.805} C_VEL
LIN {X 0,Y 418.227,Z 253.89,A -85,B 0,C 180,E1 -10220.622,E2 -10220.622} C_VEL
LIN {X 0,Y 418.248,Z 253.889,A -85,B 0,C 180,E1 -10223.972,E2 -10223.972} C_VEL
LIN {X 0,Y 418.25,Z 253.883,A -85,B 0,C 180,E1 -10227.468,E2 -10227.468} C_VEL
LIN {X 0,Y 418.267,Z 253.88,A -85,B 0,C 180,E1 -10230.893,E2 -10230.893} C_VEL
LIN {X 0,Y 418.235,Z 253.889,A -85,B 0,C 180,E1 -10234.089,E2 -10234.089} C_VEL
LIN {X 0,Y 418.234,Z 253.885,A -85,B 0,C 180,E1 -10237.259,E2 -10237.259} C_VEL
LIN {X 0,Y 418.284,Z 253.879,A -85,B 0,C 180,E1 -10240.36,E2 -10240.36} C_VEL
LIN {X 0,Y 418.316,Z 253.878,A -85,B 0,C 180,E1 -10243.4,E2 -10243.4} C_VEL
LIN {X 0,Y 418.345,Z 253.872,A -85,B 0,C 180,E1 -10246.995,E2 -10246.995} C_VEL
LIN {X 0,Y 418.331,Z 253.872,A -85,B 0,C 180,E1 -10250.323,E2 -10250.323} C_VEL
LIN {X 0,Y 418.46,Z 253.861,A -85,B 0,C 180,E1 -10253.243,E2 -10253.243} C_VEL
LIN {X 0,Y 418.316,Z 253.879,A -85,B 0,C 180,E1 -10255.176,E2 -10255.176} C_VEL
LIN {X 0,Y 418.525,Z 253.848,A -85,B 0,C 180,E1 -10258.07,E2 -10258.07} C_VEL
LIN {X 0,Y 418.656,Z 253.832,A -85,B 0,C 180,E1 -10259.994,E2 -10259.994} C_VEL
LIN {X 0,Y 418.485,Z 253.857,A -85,B 0,C 180,E1 -10262.882,E2 -10262.882} C_VEL
LIN {X 0,Y 418.45,Z 253.859,A -85,B 0,C 180,E1 -10266.605,E2 -10266.605} C_VEL
LIN {X 0,Y 418.321,Z 253.874,A -85,B 0,C 180,E1 -10269.666,E2 -10269.666} C_VEL
LIN {X 0,Y 418.326,Z 253.879,A -85,B 0,C 180,E1 -10272.994,E2 -10272.994} C_VEL
LIN {X 0,Y 418.289,Z 253.883,A -85,B 0,C 180,E1 -10276.729,E2 -10276.729} C_VEL
LIN {X 0,Y 418.244,Z 253.883,A -85,B 0,C 180,E1 -10279.784,E2 -10279.784} C_VEL
LIN {X 0,Y 418.204,Z 253.894,A -85,B 0,C 180,E1 -10282.731,E2 -10282.731} C_VEL
LIN {X 0,Y 418.237,Z 253.884,A -85,B 0,C 180,E1 -10285.898,E2 -10285.898} C_VEL
LIN {X 0,Y 418.231,Z 253.885,A -85,B 0,C 180,E1 -10289.156,E2 -10289.156} C_VEL
LIN {X 0,Y 418.22,Z 253.888,A -85,B 0,C 180,E1 -10292.838,E2 -10292.838} C_VEL
LIN {X 0,Y 418.208,Z 253.893,A -85,B 0,C 180,E1 -10296.233,E2 -10296.233} C_VEL
LIN {X 0,Y 418.221,Z 253.887,A -85,B 0,C 180,E1 -10299.675,E2 -10299.675} C_VEL
LIN {X 0,Y 418.243,Z 253.888,A -85,B 0,C 180,E1 -10302.325,E2 -10302.325} C_VEL
LIN {X 0,Y 418.229,Z 253.884,A -85,B 0,C 180,E1 -10305.109,E2 -10305.109} C_VEL
LIN {X 0,Y 418.243,Z 253.887,A -85,B 0,C 180,E1 -10307.768,E2 -10307.768} C_VEL
LIN {X 0,Y 418.215,Z 253.889,A -85,B 0,C 180,E1 -10311.555,E2 -10311.555} C_VEL
LIN {X 0,Y 418.205,Z 253.888,A -85,B 0,C 180,E1 -10315.155,E2 -10315.155} C_VEL
LIN {X 0,Y 418.189,Z 253.893,A -85,B 0,C 180,E1 -10317.468,E2 -10317.468} C_VEL
LIN {X 0,Y 418.218,Z 253.886,A -85,B 0,C 180,E1 -10320.89,E2 -10320.89} C_VEL
LIN {X 0,Y 418.214,Z 253.889,A -85,B 0,C 180,E1 -10324.093,E2 -10324.093} C_VEL
LIN {X 0,Y 418.236,Z 253.891,A -85,B 0,C 180,E1 -10327.527,E2 -10327.527} C_VEL
LIN {X 0,Y 418.255,Z 253.883,A -85,B 0,C 180,E1 -10330.363,E2 -10330.363} C_VEL
LIN {X 0,Y 418.263,Z 253.888,A -85,B 0,C 180,E1 -10333.403,E2 -10333.403} C_VEL
LIN {X 0,Y 418.292,Z 253.883,A -85,B 0,C 180,E1 -10336.992,E2 -10336.992} C_VEL
LIN {X 0,Y 418.303,Z 253.88,A -85,B 0,C 180,E1 -10340.328,E2 -10340.328} C_VEL
LIN {X 0,Y 418.451,Z 253.862,A -85,B 0,C 180,E1 -10343.248,E2 -10343.248} C_VEL
LIN {X 0,Y 418.285,Z 253.884,A -85,B 0,C 180,E1 -10345.181,E2 -10345.181} C_VEL
LIN {X 0,Y 418.48,Z 253.857,A -85,B 0,C 180,E1 -10348.075,E2 -10348.075} C_VEL
LIN {X 0,Y 418.608,Z 253.843,A -85,B 0,C 180,E1 -10350,E2 -10350} C_VEL
LIN {X 0,Y 418.454,Z 253.862,A -85,B 0,C 180,E1 -10352.888,E2 -10352.888} C_VEL
LIN {X 0,Y 418.477,Z 253.858,A -85,B 0,C 180,E1 -10355.783,E2 -10355.783} C_VEL
LIN {X 0,Y 418.352,Z 253.876,A -85,B 0,C 180,E1 -10358.696,E2 -10358.696} C_VEL
LIN {X 0,Y 418.307,Z 253.881,A -85,B 0,C 180,E1 -10362.616,E2 -10362.616} C_VEL
LIN {X 0,Y 418.272,Z 253.884,A -85,B 0,C 180,E1 -10363.309,E2 -10363.309} C_VEL
LIN {X 0,Y 417.582,Z 253.971,A -85,B 0,C 180,E1 -10364.112,E2 -10364.112} C_VEL
LIN {X 0,Y 414.703,Z 254.328,A -85,B 0,C 180,E1 -10365.418,E2 -10365.418} C_VEL
LIN {X 0,Y 412.285,Z 254.631,A -85,B 0,C 180,E1 -10366.472,E2 -10366.472} C_VEL
LIN {X 0,Y 411.259,Z 254.757,A -85,B 0,C 180,E1 -10367.287,E2 -10367.287} C_VEL
LIN {X 0,Y 411.181,Z 254.766,A -85,B 0,C 180,E1 -10367.563,E2 -10367.563} C_VEL
LIN {X 0,Y 411.181,Z 254.764,A -85,B 0,C 180,E1 -10371.034,E2 -10371.034} C_VEL
LIN {X 0,Y 411.172,Z 254.769,A -85,B 0,C 180,E1 -10374.218,E2 -10374.218} C_VEL
LIN {X 0,Y 411.201,Z 254.76,A -85,B 0,C 180,E1 -10377.481,E2 -10377.481} C_VEL
LIN {X 0,Y 411.14,Z 254.769,A -85,B 0,C 180,E1 -10380.851,E2 -10380.851} C_VEL
LIN {X 0,Y 411.151,Z 254.771,A -85,B 0,C 180,E1 -10384.338,E2 -10384.338} C_VEL
LIN {X 0,Y 411.154,Z 254.772,A -85,B 0,C 180,E1 -10387.977,E2 -10387.977} C_VEL
LIN {X 0,Y 411.16,Z 254.766,A -85,B 0,C 180,E1 -10391.241,E2 -10391.241} C_VEL
LIN {X 0,Y 411.19,Z 254.763,A -85,B 0,C 180,E1 -10394.487,E2 -10394.487} C_VEL
LIN {X 0,Y 411.188,Z 254.763,A -85,B 0,C 180,E1 -10397.302,E2 -10397.302} C_VEL
LIN {X 0,Y 411.187,Z 254.762,A -85,B 0,C 180,E1 -10400.783,E2 -10400.783} C_VEL
LIN {X 0,Y 411.16,Z 254.765,A -85,B 0,C 180,E1 -10404.477,E2 -10404.477} C_VEL
LIN {X 0,Y 411.17,Z 254.765,A -85,B 0,C 180,E1 -10406.879,E2 -10406.879} C_VEL
LIN {X 0,Y 411.181,Z 254.763,A -85,B 0,C 180,E1 -10410.655,E2 -10410.655} C_VEL
LIN {X 0,Y 411.206,Z 254.764,A -85,B 0,C 180,E1 -10413.625,E2 -10413.625} C_VEL
LIN {X 0,Y 411.168,Z 254.766,A -85,B 0,C 180,E1 -10416.858,E2 -10416.858} C_VEL
LIN {X 0,Y 411.188,Z 254.762,A -85,B 0,C 180,E1 -10420.057,E2 -10420.057} C_VEL
LIN {X 0,Y 411.24,Z 254.762,A -85,B 0,C 180,E1 -10423.137,E2 -10423.137} C_VEL
LIN {X 0,Y 411.286,Z 254.754,A -85,B 0,C 180,E1 -10426.902,E2 -10426.902} C_VEL
LIN {X 0,Y 411.273,Z 254.751,A -85,B 0,C 180,E1 -10430.167,E2 -10430.167} C_VEL
LIN {X 0,Y 411.418,Z 254.738,A -85,B 0,C 180,E1 -10433.139,E2 -10433.139} C_VEL
LIN {X 0,Y 411.442,Z 254.734,A -85,B 0,C 180,E1 -10437.069,E2 -10437.069} C_VEL
LIN {X 0,Y 411.626,Z 254.708,A -85,B 0,C 180,E1 -10440.006,E2 -10440.006} C_VEL
LIN {X 0,Y 411.427,Z 254.736,A -85,B 0,C 180,E1 -10442.943,E2 -10442.943} C_VEL
LIN {X 0,Y 411.426,Z 254.736,A -85,B 0,C 180,E1 -10446.873,E2 -10446.873} C_VEL
LIN {X 0,Y 411.284,Z 254.751,A -85,B 0,C 180,E1 -10449.844,E2 -10449.844} C_VEL
LIN {X 0,Y 411.304,Z 254.748,A -85,B 0,C 180,E1 -10453.109,E2 -10453.109} C_VEL
LIN {X 0,Y 411.258,Z 254.754,A -85,B 0,C 180,E1 -10456.894,E2 -10456.894} C_VEL
LIN {X 0,Y 411.233,Z 254.76,A -85,B 0,C 180,E1 -10459.991,E2 -10459.991} C_VEL
LIN {X 0,Y 411.198,Z 254.76,A -85,B 0,C 180,E1 -10463.153,E2 -10463.153} C_VEL
LIN {X 0,Y 411.185,Z 254.766,A -85,B 0,C 180,E1 -10466.389,E2 -10466.389} C_VEL
LIN {X 0,Y 411.203,Z 254.763,A -85,B 0,C 180,E1 -10469.717,E2 -10469.717} C_VEL
LIN {X 0,Y 411.212,Z 254.759,A -85,B 0,C 180,E1 -10473.16,E2 -10473.16} C_VEL
LIN {X 0,Y 411.199,Z 254.765,A -85,B 0,C 180,E1 -10476.556,E2 -10476.556} C_VEL
LIN {X 0,Y 411.197,Z 254.767,A -85,B 0,C 180,E1 -10479.231,E2 -10479.231} C_VEL
LIN {X 0,Y 411.677,Z 258.069,A -85,B 0,C 180,E1 -10482.772,E2 -10482.772} C_VEL
LIN {X 0,Y 412.059,Z 261.142,A -85,B 0,C 180,E1 -10485.758,E2 -10485.758} C_VEL
LIN {X 0,Y 412.159,Z 264.013,A -85,B 0,C 180,E1 -10488.318,E2 -10488.318} C_VEL
LIN {X 0,Y 411.917,Z 268.096,A -85,B 0,C 180,E1 -10491.71,E2 -10491.71} C_VEL
LIN {X 0,Y 411.551,Z 272.433,A -85,B 0,C 180,E1 -10495.059,E2 -10495.059} C_VEL
LIN {X 0,Y 411.244,Z 276.476,A -85,B 0,C 180,E1 -10498.01,E2 -10498.01} C_VEL
LIN {X 0,Y 410.845,Z 281.295,A -85,B 0,C 180,E1 -10501.382,E2 -10501.382} C_VEL
LIN {X 0,Y 410.546,Z 286.908,A -85,B 0,C 180,E1 -10505.139,E2 -10505.139} C_VEL
LIN {X 0,Y 410.343,Z 291.137,A -85,B 0,C 180,E1 -10507.865,E2 -10507.865} C_VEL
LIN {X 0,Y 410.145,Z 296.122,A -85,B 0,C 180,E1 -10511,E2 -10511} C_VEL
LIN {X 0,Y 410.091,Z 298.367,A -85,B 0,C 180,E1 -10512.42,E2 -10512.42} C_VEL
LIN {X 0,Y 413.061,Z 314.37,A -85,B 0,C 180,E1 -10513.108,E2 -10513.108} C_VEL
LIN {X 0,Y 414.482,Z 325.034,A -85,B 0,C 180,E1 -10513.714,E2 -10513.714} C_VEL
LIN {X 0,Y 414.458,Z 332,A -85,B 0,C 180,E1 -10514.149,E2 -10514.149} C_VEL
LIN {X 0,Y 413.573,Z 344.475,A -85,B 0,C 180,E1 -10515.107,E2 -10515.107} C_VEL
LIN {X 0,Y 412.943,Z 353.408,A -85,B 0,C 180,E1 -10515.963,E2 -10515.963} C_VEL
LIN {X 0,Y 412.342,Z 361.954,A -85,B 0,C 180,E1 -10516.948,E2 -10516.948} C_VEL
LIN {X 0,Y 411.814,Z 369.175,A -85,B 0,C 180,E1 -10517.933,E2 -10517.933} C_VEL
LIN {X 0,Y 411.315,Z 375.377,A -85,B 0,C 180,E1 -10518.918,E2 -10518.918} C_VEL
LIN {X 0,Y 410.829,Z 381.914,A -85,B 0,C 180,E1 -10520.15,E2 -10520.15} C_VEL
LIN {X 0,Y 410.541,Z 386.416,A -85,B 0,C 180,E1 -10521.137,E2 -10521.137} C_VEL
LIN {X 0,Y 410.213,Z 391.907,A -85,B 0,C 180,E1 -10522.618,E2 -10522.618} C_VEL
LIN {X 0,Y 410.027,Z 396.23,A -85,B 0,C 180,E1 -10524.097,E2 -10524.097} C_VEL
LIN {X 0,Y 410.026,Z 398.598,A -85,B 0,C 180,E1 -10525.084,E2 -10525.084} C_VEL
LIN {X 0,Y 409.922,Z 401.781,A -85,B 0,C 180,E1 -10527.052,E2 -10527.052} C_VEL
LIN {X 0,Y 409.972,Z 402.839,A -85,B 0,C 180,E1 -10528.035,E2 -10528.035} C_VEL
LIN {X 0,Y 409.926,Z 403.426,A -85,B 0,C 180,E1 -10529.018,E2 -10529.018} C_VEL
LIN {X 0,Y 409.926,Z 403.426,A -85,B 0,C 180,E1 -10530.982,E2 -10530.982} C_VEL
LIN {X 0,Y 409.972,Z 402.839,A -85,B 0,C 180,E1 -10531.965,E2 -10531.965} C_VEL
LIN {X 0,Y 409.925,Z 400.394,A -85,B 0,C 180,E1 -10533.932,E2 -10533.932} C_VEL
LIN {X 0,Y 410.024,Z 397.448,A -85,B 0,C 180,E1 -10535.409,E2 -10535.409} C_VEL
LIN {X 0,Y 410.18,Z 393.462,A -85,B 0,C 180,E1 -10536.888,E2 -10536.888} C_VEL
LIN {X 0,Y 410.428,Z 388.332,A -85,B 0,C 180,E1 -10538.369,E2 -10538.369} C_VEL
LIN {X 0,Y 410.754,Z 383.07,A -85,B 0,C 180,E1 -10539.603,E2 -10539.603} C_VEL
LIN {X 0,Y 411.173,Z 376.752,A -85,B 0,C 180,E1 -10540.837,E2 -10540.837} C_VEL
LIN {X 0,Y 411.668,Z 370.801,A -85,B 0,C 180,E1 -10541.821,E2 -10541.821} C_VEL
LIN {X 0,Y 412.219,Z 363.874,A -85,B 0,C 180,E1 -10542.805,E2 -10542.805} C_VEL
LIN {X 0,Y 412.814,Z 355.693,A -85,B 0,C 180,E1 -10543.789,E2 -10543.789} C_VEL
LIN {X 0,Y 413.325,Z 347.313,A -85,B 0,C 180,E1 -10544.638,E2 -10544.638} C_VEL
LIN {X 0,Y 413.959,Z 338.461,A -85,B 0,C 180,E1 -10545.383,E2 -10545.383} C_VEL
LIN {X 0,Y 414.681,Z 328.526,A -85,B 0,C 180,E1 -10546.06,E2 -10546.06} C_VEL
LIN {X 0,Y 413.893,Z 319.969,A -85,B 0,C 180,E1 -10546.582,E2 -10546.582} C_VEL
LIN {X 0,Y 412.111,Z 308.943,A -85,B 0,C 180,E1 -10547.142,E2 -10547.142} C_VEL
LIN {X 0,Y 410.089,Z 298.367,A -85,B 0,C 180,E1 -10547.58,E2 -10547.58} C_VEL
LIN {X 0,Y 410.264,Z 292.775,A -85,B 0,C 180,E1 -10551.084,E2 -10551.084} C_VEL
LIN {X 0,Y 410.495,Z 287.822,A -85,B 0,C 180,E1 -10554.261,E2 -10554.261} C_VEL
LIN {X 0,Y 410.735,Z 282.913,A -85,B 0,C 180,E1 -10557.515,E2 -10557.515} C_VEL
LIN {X 0,Y 411.151,Z 278.059,A -85,B 0,C 180,E1 -10560.85,E2 -10560.85} C_VEL
LIN {X 0,Y 411.483,Z 273.28,A -85,B 0,C 180,E1 -10564.306,E2 -10564.306} C_VEL
LIN {X 0,Y 411.754,Z 270.138,A -85,B 0,C 180,E1 -10566.683,E2 -10566.683} C_VEL
LIN {X 0,Y 412.023,Z 266.144,A -85,B 0,C 180,E1 -10569.858,E2 -10569.858} C_VEL
LIN {X 0,Y 412.179,Z 262.663,A -85,B 0,C 180,E1 -10572.841,E2 -10572.841} C_VEL
LIN {X 0,Y 411.857,Z 259.519,A -85,B 0,C 180,E1 -10575.781,E2 -10575.781} C_VEL
LIN {X 0,Y 411.347,Z 255.893,A -85,B 0,C 180,E1 -10579.511,E2 -10579.511} C_VEL
LIN {X 0,Y 411.197,Z 254.766,A -85,B 0,C 180,E1 -10580.769,E2 -10580.769} C_VEL
LIN {X 0,Y 411.201,Z 254.769,A -85,B 0,C 180,E1 -10584.467,E2 -10584.467} C_VEL
LIN {X 0,Y 411.213,Z 254.759,A -85,B 0,C 180,E1 -10586.87,E2 -10586.87} C_VEL
LIN {X 0,Y 411.217,Z 254.759,A -85,B 0,C 180,E1 -10590.646,E2 -10590.646} C_VEL
LIN {X 0,Y 411.185,Z 254.766,A -85,B 0,C 180,E1 -10593.611,E2 -10593.611} C_VEL
LIN {X 0,Y 411.198,Z 254.76,A -85,B 0,C 180,E1 -10596.847,E2 -10596.847} C_VEL
LIN {X 0,Y 411.216,Z 254.762,A -85,B 0,C 180,E1 -10600.046,E2 -10600.046} C_VEL
LIN {X 0,Y 411.264,Z 254.754,A -85,B 0,C 180,E1 -10603.126,E2 -10603.126} C_VEL
LIN {X 0,Y 411.304,Z 254.748,A -85,B 0,C 180,E1 -10606.891,E2 -10606.891} C_VEL
LIN {X 0,Y 411.284,Z 254.751,A -85,B 0,C 180,E1 -10610.156,E2 -10610.156} C_VEL
LIN {X 0,Y 411.426,Z 254.736,A -85,B 0,C 180,E1 -10613.127,E2 -10613.127} C_VEL
LIN {X 0,Y 411.289,Z 254.753,A -85,B 0,C 180,E1 -10615.093,E2 -10615.093} C_VEL
LIN {X 0,Y 411.494,Z 254.724,A -85,B 0,C 180,E1 -10618.037,E2 -10618.037} C_VEL
LIN {X 0,Y 411.626,Z 254.708,A -85,B 0,C 180,E1 -10619.994,E2 -10619.994} C_VEL
LIN {X 0,Y 411.442,Z 254.734,A -85,B 0,C 180,E1 -10622.931,E2 -10622.931} C_VEL
LIN {X 0,Y 411.418,Z 254.738,A -85,B 0,C 180,E1 -10626.861,E2 -10626.861} C_VEL
LIN {X 0,Y 411.273,Z 254.751,A -85,B 0,C 180,E1 -10629.833,E2 -10629.833} C_VEL
LIN {X 0,Y 411.286,Z 254.754,A -85,B 0,C 180,E1 -10633.098,E2 -10633.098} C_VEL
LIN {X 0,Y 411.234,Z 254.762,A -85,B 0,C 180,E1 -10636.883,E2 -10636.883} C_VEL
LIN {X 0,Y 411.205,Z 254.76,A -85,B 0,C 180,E1 -10639.981,E2 -10639.981} C_VEL
LIN {X 0,Y 411.168,Z 254.766,A -85,B 0,C 180,E1 -10643.142,E2 -10643.142} C_VEL
LIN {X 0,Y 411.206,Z 254.764,A -85,B 0,C 180,E1 -10646.375,E2 -10646.375} C_VEL
LIN {X 0,Y 411.166,Z 254.765,A -85,B 0,C 180,E1 -10649.707,E2 -10649.707} C_VEL
LIN {X 0,Y 411.169,Z 254.764,A -85,B 0,C 180,E1 -10653.15,E2 -10653.15} C_VEL
LIN {X 0,Y 411.155,Z 254.77,A -85,B 0,C 180,E1 -10656.547,E2 -10656.547} C_VEL
LIN {X 0,Y 411.184,Z 254.764,A -85,B 0,C 180,E1 -10659.725,E2 -10659.725} C_VEL
LIN {X 0,Y 411.184,Z 254.762,A -85,B 0,C 180,E1 -10663.121,E2 -10663.121} C_VEL
LIN {X 0,Y 411.193,Z 254.765,A -85,B 0,C 180,E1 -10665.866,E2 -10665.866} C_VEL
LIN {X 0,Y 411.164,Z 254.766,A -85,B 0,C 180,E1 -10669.495,E2 -10669.495} C_VEL
LIN {X 0,Y 411.153,Z 254.772,A -85,B 0,C 180,E1 -10672.023,E2 -10672.023} C_VEL
LIN {X 0,Y 411.151,Z 254.771,A -85,B 0,C 180,E1 -10675.662,E2 -10675.662} C_VEL
LIN {X 0,Y 411.14,Z 254.769,A -85,B 0,C 180,E1 -10679.149,E2 -10679.149} C_VEL
LIN {X 0,Y 411.201,Z 254.76,A -85,B 0,C 180,E1 -10682.519,E2 -10682.519} C_VEL
LIN {X 0,Y 411.172,Z 254.769,A -85,B 0,C 180,E1 -10685.782,E2 -10685.782} C_VEL
LIN {X 0,Y 411.181,Z 254.764,A -85,B 0,C 180,E1 -10688.966,E2 -10688.966} C_VEL
LIN {X 0,Y 411.193,Z 254.766,A -85,B 0,C 180,E1 -10692.083,E2 -10692.083} C_VEL
LIN {X 0,Y 411.209,Z 254.765,A -85,B 0,C 180,E1 -10695.146,E2 -10695.146} C_VEL
LIN {X 0,Y 411.238,Z 254.758,A -85,B 0,C 180,E1 -10698.166,E2 -10698.166} C_VEL
LIN {X 0,Y 411.417,Z 254.738,A -85,B 0,C 180,E1 -10702.146,E2 -10702.146} C_VEL
LIN {X 0,Y 411.436,Z 254.735,A -85,B 0,C 180,E1 -10704.118,E2 -10704.118} C_VEL
LIN {X 0,Y 411.449,Z 254.733,A -85,B 0,C 180,E1 -10708.042,E2 -10708.042} C_VEL
LIN {X 0,Y 411.578,Z 254.719,A -85,B 0,C 180,E1 -10710,E2 -10710} C_VEL
LIN {X 0,Y 411.409,Z 254.739,A -85,B 0,C 180,E1 -10712.938,E2 -10712.938} C_VEL
LIN {X 0,Y 411.436,Z 254.735,A -85,B 0,C 180,E1 -10715.882,E2 -10715.882} C_VEL
LIN {X 0,Y 411.304,Z 254.754,A -85,B 0,C 180,E1 -10718.846,E2 -10718.846} C_VEL
LIN {X 0,Y 411.238,Z 254.758,A -85,B 0,C 180,E1 -10721.834,E2 -10721.834} C_VEL
LIN {X 0,Y 411.209,Z 254.765,A -85,B 0,C 180,E1 -10724.854,E2 -10724.854} C_VEL
LIN {X 0,Y 411.181,Z 254.766,A -85,B 0,C 180,E1 -10727.563,E2 -10727.563} C_VEL
LIN {X 0,Y 410.524,Z 254.851,A -85,B 0,C 180,E1 -10728.381,E2 -10728.381} C_VEL
LIN {X 0,Y 407.662,Z 255.204,A -85,B 0,C 180,E1 -10729.711,E2 -10729.711} C_VEL
LIN {X 0,Y 405.24,Z 255.506,A -85,B 0,C 180,E1 -10730.784,E2 -10730.784} C_VEL
LIN {X 0,Y 404.211,Z 255.631,A -85,B 0,C 180,E1 -10731.615,E2 -10731.615} C_VEL
LIN {X 0,Y 404.134,Z 255.641,A -85,B 0,C 180,E1 -10731.896,E2 -10731.896} C_VEL
LIN {X 0,Y 404.157,Z 255.638,A -85,B 0,C 180,E1 -10735.3,E2 -10735.3} C_VEL
LIN {X 0,Y 404.14,Z 255.643,A -85,B 0,C 180,E1 -10738.003,E2 -10738.003} C_VEL
LIN {X 0,Y 404.086,Z 255.647,A -85,B 0,C 180,E1 -10741.562,E2 -10741.562} C_VEL
LIN {X 0,Y 404.131,Z 255.641,A -85,B 0,C 180,E1 -10745.02,E2 -10745.02} C_VEL
LIN {X 0,Y 404.113,Z 255.644,A -85,B 0,C 180,E1 -10748.76,E2 -10748.76} C_VEL
LIN {X 0,Y 404.142,Z 255.642,A -85,B 0,C 180,E1 -10751.615,E2 -10751.615} C_VEL
LIN {X 0,Y 404.155,Z 255.639,A -85,B 0,C 180,E1 -10754.535,E2 -10754.535} C_VEL
LIN {X 0,Y 404.166,Z 255.638,A -85,B 0,C 180,E1 -10757.311,E2 -10757.311} C_VEL
LIN {X 0,Y 404.127,Z 255.646,A -85,B 0,C 180,E1 -10759.961,E2 -10759.961} C_VEL
LIN {X 0,Y 404.1,Z 255.646,A -85,B 0,C 180,E1 -10763.13,E2 -10763.13} C_VEL
LIN {X 0,Y 404.108,Z 255.645,A -85,B 0,C 180,E1 -10766.194,E2 -10766.194} C_VEL
LIN {X 0,Y 404.111,Z 255.648,A -85,B 0,C 180,E1 -10769.721,E2 -10769.721} C_VEL
LIN {X 0,Y 404.164,Z 255.64,A -85,B 0,C 180,E1 -10773.129,E2 -10773.129} C_VEL
LIN {X 0,Y 404.145,Z 255.646,A -85,B 0,C 180,E1 -10775.34,E2 -10775.34} C_VEL
LIN {X 0,Y 404.111,Z 255.644,A -85,B 0,C 180,E1 -10778.587,E2 -10778.587} C_VEL
LIN {X 0,Y 404.18,Z 255.636,A -85,B 0,C 180,E1 -10781.768,E2 -10781.768} C_VEL
LIN {X 0,Y 404.183,Z 255.638,A -85,B 0,C 180,E1 -10784.888,E2 -10784.888} C_VEL
LIN {X 0,Y 404.237,Z 255.628,A -85,B 0,C 180,E1 -10787.965,E2 -10787.965} C_VEL
LIN {X 0,Y 404.249,Z 255.633,A -85,B 0,C 180,E1 -10791.005,E2 -10791.005} C_VEL
LIN {X 0,Y 404.381,Z 255.61,A -85,B 0,C 180,E1 -10794.021,E2 -10794.021} C_VEL
LIN {X 0,Y 404.468,Z 255.599,A -85,B 0,C 180,E1 -10798.014,E2 -10798.014} C_VEL
LIN {X 0,Y 404.596,Z 255.583,A -85,B 0,C 180,E1 -10800.006,E2 -10800.006} C_VEL
LIN {X 0,Y 404.387,Z 255.612,A -85,B 0,C 180,E1 -10802.994,E2 -10802.994} C_VEL
LIN {X 0,Y 404.376,Z 255.613,A -85,B 0,C 180,E1 -10806.993,E2 -10806.993} C_VEL
LIN {X 0,Y 404.246,Z 255.628,A -85,B 0,C 180,E1 -10811.03,E2 -10811.03} C_VEL
LIN {X 0,Y 404.208,Z 255.635,A -85,B 0,C 180,E1 -10814.094,E2 -10814.094} C_VEL
LIN {X 0,Y 404.203,Z 255.632,A -85,B 0,C 180,E1 -10817.198,E2 -10817.198} C_VEL
LIN {X 0,Y 404.166,Z 255.642,A -85,B 0,C 180,E1 -10820.356,E2 -10820.356} C_VEL
LIN {X 0,Y 404.16,Z 255.638,A -85,B 0,C 180,E1 -10823.58,E2 -10823.58} C_VEL
LIN {X 0,Y 404.129,Z 255.641,A -85,B 0,C 180,E1 -10826.887,E2 -10826.887} C_VEL
LIN {X 0,Y 404.15,Z 255.642,A -85,B 0,C 180,E1 -10830.289,E2 -10830.289} C_VEL
LIN {X 0,Y 404.148,Z 255.644,A -85,B 0,C 180,E1 -10833.817,E2 -10833.817} C_VEL
LIN {X 0,Y 404.142,Z 255.644,A -85,B 0,C 180,E1 -10836.878,E2 -10836.878} C_VEL
LIN {X 0,Y 404.147,Z 255.646,A -85,B 0,C 180,E1 -10838.762,E2 -10838.762} C_VEL
LIN {X 0,Y 404.523,Z 258.121,A -85,B 0,C 180,E1 -10841.665,E2 -10841.665} C_VEL
LIN {X 0,Y 404.894,Z 261.032,A -85,B 0,C 180,E1 -10844.631,E2 -10844.631} C_VEL
LIN {X 0,Y 405.14,Z 264.006,A -85,B 0,C 180,E1 -10847.428,E2 -10847.428} C_VEL
LIN {X 0,Y 404.984,Z 267.042,A -85,B 0,C 180,E1 -10850.053,E2 -10850.053} C_VEL
LIN {X 0,Y 404.727,Z 270.692,A -85,B 0,C 180,E1 -10853.019,E2 -10853.019} C_VEL
LIN {X 0,Y 404.369,Z 275.263,A -85,B 0,C 180,E1 -10856.543,E2 -10856.543} C_VEL
LIN {X 0,Y 403.99,Z 279.604,A -85,B 0,C 180,E1 -10859.703,E2 -10859.703} C_VEL
LIN {X 0,Y 403.618,Z 284.453,A -85,B 0,C 180,E1 -10863.082,E2 -10863.082} C_VEL
LIN {X 0,Y 403.337,Z 289.355,A -85,B 0,C 180,E1 -10866.374,E2 -10866.374} C_VEL
LIN {X 0,Y 403.14,Z 294.316,A -85,B 0,C 180,E1 -10869.595,E2 -10869.595} C_VEL
LIN {X 0,Y 403.016,Z 298.217,A -85,B 0,C 180,E1 -10872.125,E2 -10872.125} C_VEL
LIN {X 0,Y 405.102,Z 308.691,A -85,B 0,C 180,E1 -10872.55,E2 -10872.55} C_VEL
LIN {X 0,Y 406.644,Z 318.251,A -85,B 0,C 180,E1 -10873.037,E2 -10873.037} C_VEL
LIN {X 0,Y 407.704,Z 327.03,A -85,B 0,C 180,E1 -10873.575,E2 -10873.575} C_VEL
LIN {X 0,Y 407.405,Z 335.004,A -85,B 0,C 180,E1 -10874.107,E2 -10874.107} C_VEL
LIN {X 0,Y 406.71,Z 344.28,A -85,B 0,C 180,E1 -10874.849,E2 -10874.849} C_VEL
LIN {X 0,Y 406.031,Z 353.231,A -85,B 0,C 180,E1 -10875.721,E2 -10875.721} C_VEL
LIN {X 0,Y 405.383,Z 361.758,A -85,B 0,C 180,E1 -10876.72,E2 -10876.72} C_VEL
LIN {X 0,Y 404.828,Z 368.979,A -85,B 0,C 180,E1 -10877.722,E2 -10877.722} C_VEL
LIN {X 0,Y 404.318,Z 375.181,A -85,B 0,C 180,E1 -10878.723,E2 -10878.723} C_VEL
LIN {X 0,Y 403.825,Z 381.719,A -85,B 0,C 180,E1 -10879.978,E2 -10879.978} C_VEL
LIN {X 0,Y 403.497,Z 386.221,A -85,B 0,C 180,E1 -10880.981,E2 -10880.981} C_VEL
LIN {X 0,Y 403.158,Z 391.712,A -85,B 0,C 180,E1 -10882.488,E2 -10882.488} C_VEL
LIN {X 0,Y 402.953,Z 396.035,A -85,B 0,C 180,E1 -10883.993,E2 -10883.993} C_VEL
LIN {X 0,Y 402.938,Z 398.403,A -85,B 0,C 180,E1 -10884.997,E2 -10884.997} C_VEL
LIN {X 0,Y 402.847,Z 400.199,A -85,B 0,C 180,E1 -10885.999,E2 -10885.999} C_VEL
LIN {X 0,Y 402.87,Z 402.644,A -85,B 0,C 180,E1 -10888.001,E2 -10888.001} C_VEL
LIN {X 0,Y 402.854,Z 403.232,A -85,B 0,C 180,E1 -10889,E2 -10889} C_VEL
LIN {X 0,Y 402.854,Z 403.232,A -85,B 0,C 180,E1 -10891,E2 -10891} C_VEL
LIN {X 0,Y 402.87,Z 402.644,A -85,B 0,C 180,E1 -10891.999,E2 -10891.999} C_VEL
LIN {X 0,Y 402.847,Z 400.199,A -85,B 0,C 180,E1 -10894.001,E2 -10894.001} C_VEL
LIN {X 0,Y 402.923,Z 397.252,A -85,B 0,C 180,E1 -10895.505,E2 -10895.505} C_VEL
LIN {X 0,Y 403.093,Z 393.266,A -85,B 0,C 180,E1 -10897.01,E2 -10897.01} C_VEL
LIN {X 0,Y 403.369,Z 388.136,A -85,B 0,C 180,E1 -10898.516,E2 -10898.516} C_VEL
LIN {X 0,Y 403.719,Z 382.874,A -85,B 0,C 180,E1 -10899.772,E2 -10899.772} C_VEL
LIN {X 0,Y 404.168,Z 376.556,A -85,B 0,C 180,E1 -10901.027,E2 -10901.027} C_VEL
LIN {X 0,Y 404.692,Z 370.606,A -85,B 0,C 180,E1 -10902.028,E2 -10902.028} C_VEL
LIN {X 0,Y 405.248,Z 363.678,A -85,B 0,C 180,E1 -10903.029,E2 -10903.029} C_VEL
LIN {X 0,Y 405.868,Z 355.497,A -85,B 0,C 180,E1 -10904.029,E2 -10904.029} C_VEL
LIN {X 0,Y 406.443,Z 347.118,A -85,B 0,C 180,E1 -10904.891,E2 -10904.891} C_VEL
LIN {X 0,Y 407.082,Z 338.266,A -85,B 0,C 180,E1 -10905.649,E2 -10905.649} C_VEL
LIN {X 0,Y 407.802,Z 328.663,A -85,B 0,C 180,E1 -10906.317,E2 -10906.317} C_VEL
LIN {X 0,Y 406.859,Z 319.768,A -85,B 0,C 180,E1 -10906.878,E2 -10906.878} C_VEL
LIN {X 0,Y 405.151,Z 309.281,A -85,B 0,C 180,E1 -10907.426,E2 -10907.426} C_VEL
LIN {X 0,Y 402.996,Z 298.183,A -85,B 0,C 180,E1 -10907.897,E2 -10907.897} C_VEL
LIN {X 0,Y 403.14,Z 294.272,A -85,B 0,C 180,E1 -10910.405,E2 -10910.405} C_VEL
LIN {X 0,Y 403.34,Z 289.34,A -85,B 0,C 180,E1 -10913.625,E2 -10913.625} C_VEL
LIN {X 0,Y 403.618,Z 284.443,A -85,B 0,C 180,E1 -10916.918,E2 -10916.918} C_VEL
LIN {X 0,Y 403.993,Z 279.594,A -85,B 0,C 180,E1 -10920.297,E2 -10920.297} C_VEL
LIN {X 0,Y 404.369,Z 275.258,A -85,B 0,C 180,E1 -10923.457,E2 -10923.457} C_VEL
LIN {X 0,Y 404.722,Z 270.662,A -85,B 0,C 180,E1 -10926.98,E2 -10926.98} C_VEL
LIN {X 0,Y 405.031,Z 266.69,A -85,B 0,C 180,E1 -10930.224,E2 -10930.224} C_VEL
LIN {X 0,Y 405.142,Z 264.003,A -85,B 0,C 180,E1 -10932.572,E2 -10932.572} C_VEL
LIN {X 0,Y 404.894,Z 261.027,A -85,B 0,C 180,E1 -10935.369,E2 -10935.369} C_VEL
LIN {X 0,Y 404.478,Z 257.8,A -85,B 0,C 180,E1 -10938.675,E2 -10938.675} C_VEL
LIN {X 0,Y 404.15,Z 255.644,A -85,B 0,C 180,E1 -10941.491,E2 -10941.491} C_VEL
LIN {X 0,Y 404.185,Z 255.64,A -85,B 0,C 180,E1 -10944.979,E2 -10944.979} C_VEL
LIN {X 0,Y 404.145,Z 255.641,A -85,B 0,C 180,E1 -10948.438,E2 -10948.438} C_VEL
LIN {X 0,Y 404.16,Z 255.637,A -85,B 0,C 180,E1 -10950.859,E2 -10950.859} C_VEL
LIN {X 0,Y 404.148,Z 255.642,A -85,B 0,C 180,E1 -10954.226,E2 -10954.226} C_VEL
LIN {X 0,Y 404.171,Z 255.639,A -85,B 0,C 180,E1 -10957.503,E2 -10957.503} C_VEL
LIN {X 0,Y 404.163,Z 255.637,A -85,B 0,C 180,E1 -10960.703,E2 -10960.703} C_VEL
LIN {X 0,Y 404.221,Z 255.634,A -85,B 0,C 180,E1 -10963.843,E2 -10963.843} C_VEL
LIN {X 0,Y 404.282,Z 255.623,A -85,B 0,C 180,E1 -10966.934,E2 -10966.934} C_VEL
LIN {X 0,Y 404.25,Z 255.628,A -85,B 0,C 180,E1 -10969.983,E2 -10969.983} C_VEL
LIN {X 0,Y 404.376,Z 255.613,A -85,B 0,C 180,E1 -10973.007,E2 -10973.007} C_VEL
LIN {X 0,Y 404.261,Z 255.628,A -85,B 0,C 180,E1 -10975.008,E2 -10975.008} C_VEL
LIN {X 0,Y 404.463,Z 255.6,A -85,B 0,C 180,E1 -10978.003,E2 -10978.003} C_VEL
LIN {X 0,Y 404.596,Z 255.583,A -85,B 0,C 180,E1 -10979.994,E2 -10979.994} C_VEL
LIN {X 0,Y 404.4,Z 255.612,A -85,B 0,C 180,E1 -10982.983,E2 -10982.983} C_VEL
LIN {X 0,Y 404.368,Z 255.617,A -85,B 0,C 180,E1 -10986.982,E2 -10986.982} C_VEL
LIN {X 0,Y 404.233,Z 255.635,A -85,B 0,C 180,E1 -10991.019,E2 -10991.019} C_VEL
LIN {X 0,Y 404.189,Z 255.634,A -85,B 0,C 180,E1 -10994.082,E2 -10994.082} C_VEL
LIN {X 0,Y 404.179,Z 255.638,A -85,B 0,C 180,E1 -10997.186,E2 -10997.186} C_VEL
LIN {X 0,Y 404.138,Z 255.643,A -85,B 0,C 180,E1 -11000.345,E2 -11000.345} C_VEL
LIN {X 0,Y 404.135,Z 255.64,A -85,B 0,C 180,E1 -11003.569,E2 -11003.569} C_VEL
LIN {X 0,Y 404.153,Z 255.638,A -85,B 0,C 180,E1 -11005.76,E2 -11005.76} C_VEL
LIN {X 0,Y 404.163,Z 255.638,A -85,B 0,C 180,E1 -11007.994,E2 -11007.994} C_VEL
LIN {X 0,Y 404.103,Z 255.644,A -85,B 0,C 180,E1 -11011.552,E2 -11011.552} C_VEL
LIN {X 0,Y 404.146,Z 255.64,A -85,B 0,C 180,E1 -11015.01,E2 -11015.01} C_VEL
LIN {X 0,Y 404.121,Z 255.644,A -85,B 0,C 180,E1 -11018.75,E2 -11018.75} C_VEL
LIN {X 0,Y 404.148,Z 255.64,A -85,B 0,C 180,E1 -11021.605,E2 -11021.605} C_VEL
LIN {X 0,Y 404.162,Z 255.64,A -85,B 0,C 180,E1 -11024.526,E2 -11024.526} C_VEL
LIN {X 0,Y 404.162,Z 255.637,A -85,B 0,C 180,E1 -11027.3,E2 -11027.3} C_VEL
LIN {X 0,Y 404.119,Z 255.649,A -85,B 0,C 180,E1 -11029.951,E2 -11029.951} C_VEL
LIN {X 0,Y 404.088,Z 255.646,A -85,B 0,C 180,E1 -11033.12,E2 -11033.12} C_VEL
LIN {X 0,Y 404.09,Z 255.649,A -85,B 0,C 180,E1 -11036.183,E2 -11036.183} C_VEL
LIN {X 0,Y 404.096,Z 255.652,A -85,B 0,C 180,E1 -11039.712,E2 -11039.712} C_VEL
LIN {X 0,Y 404.137,Z 255.641,A -85,B 0,C 180,E1 -11043.119,E2 -11043.119} C_VEL
LIN {X 0,Y 404.125,Z 255.642,A -85,B 0,C 180,E1 -11046.423,E2 -11046.423} C_VEL
LIN {X 0,Y 404.166,Z 255.643,A -85,B 0,C 180,E1 -11049.858,E2 -11049.858} C_VEL
LIN {X 0,Y 404.156,Z 255.644,A -85,B 0,C 180,E1 -11052.989,E2 -11052.989} C_VEL
LIN {X 0,Y 404.203,Z 255.638,A -85,B 0,C 180,E1 -11056.787,E2 -11056.787} C_VEL
LIN {X 0,Y 404.211,Z 255.636,A -85,B 0,C 180,E1 -11059.987,E2 -11059.987} C_VEL
LIN {X 0,Y 404.38,Z 255.615,A -85,B 0,C 180,E1 -11063.012,E2 -11063.012} C_VEL
LIN {X 0,Y 404.229,Z 255.636,A -85,B 0,C 180,E1 -11065.013,E2 -11065.013} C_VEL
LIN {X 0,Y 404.419,Z 255.609,A -85,B 0,C 180,E1 -11068.008,E2 -11068.008} C_VEL
LIN {X 0,Y 404.548,Z 255.595,A -85,B 0,C 180,E1 -11070,E2 -11070} C_VEL
LIN {X 0,Y 404.367,Z 255.616,A -85,B 0,C 180,E1 -11072.989,E2 -11072.989} C_VEL
LIN {X 0,Y 404.38,Z 255.615,A -85,B 0,C 180,E1 -11076.988,E2 -11076.988} C_VEL
LIN {X 0,Y 404.211,Z 255.636,A -85,B 0,C 180,E1 -11080.013,E2 -11080.013} C_VEL
LIN {X 0,Y 404.203,Z 255.638,A -85,B 0,C 180,E1 -11083.213,E2 -11083.213} C_VEL
LIN {X 0,Y 404.156,Z 255.644,A -85,B 0,C 180,E1 -11087.011,E2 -11087.011} C_VEL
LIN {X 0,Y 404.146,Z 255.645,A -85,B 0,C 180,E1 -11090.352,E2 -11090.352} C_VEL
LIN {X 0,Y 404.134,Z 255.641,A -85,B 0,C 180,E1 -11091.896,E2 -11091.896} C_VEL
LIN {X 0,Y 403.483,Z 255.729,A -85,B 0,C 180,E1 -11092.727,E2 -11092.727} C_VEL
LIN {X 0,Y 400.63,Z 256.091,A -85,B 0,C 180,E1 -11094.078,E2 -11094.078} C_VEL
LIN {X 0,Y 398.204,Z 256.394,A -85,B 0,C 180,E1 -11095.169,E2 -11095.169} C_VEL
LIN {X 0,Y 397.161,Z 256.518,A -85,B 0,C 180,E1 -11096.013,E2 -11096.013} C_VEL
LIN {X 0,Y 397.077,Z 256.525,A -85,B 0,C 180,E1 -11096.299,E2 -11096.299} C_VEL
LIN {X 0,Y 397.069,Z 256.525,A -85,B 0,C 180,E1 -11098.547,E2 -11098.547} C_VEL
LIN {X 0,Y 397.025,Z 256.532,A -85,B 0,C 180,E1 -11102.076,E2 -11102.076} C_VEL
LIN {X 0,Y 397.066,Z 256.522,A -85,B 0,C 180,E1 -11105.508,E2 -11105.508} C_VEL
LIN {X 0,Y 397.087,Z 256.518,A -85,B 0,C 180,E1 -11108.868,E2 -11108.868} C_VEL
LIN {X 0,Y 397.112,Z 256.519,A -85,B 0,C 180,E1 -11112.26,E2 -11112.26} C_VEL
LIN {X 0,Y 397.108,Z 256.516,A -85,B 0,C 180,E1 -11115.064,E2 -11115.064} C_VEL
LIN {X 0,Y 397.113,Z 256.52,A -85,B 0,C 180,E1 -11118.012,E2 -11118.012} C_VEL
LIN {X 0,Y 397.068,Z 256.528,A -85,B 0,C 180,E1 -11121.731,E2 -11121.731} C_VEL
LIN {X 0,Y 397.088,Z 256.524,A -85,B 0,C 180,E1 -11125.513,E2 -11125.513} C_VEL
LIN {X 0,Y 397.043,Z 256.526,A -85,B 0,C 180,E1 -11129.123,E2 -11129.123} C_VEL
LIN {X 0,Y 397.162,Z 256.509,A -85,B 0,C 180,E1 -11132.616,E2 -11132.616} C_VEL
LIN {X 0,Y 397.1,Z 256.518,A -85,B 0,C 180,E1 -11135.988,E2 -11135.988} C_VEL
LIN {X 0,Y 397.113,Z 256.517,A -85,B 0,C 180,E1 -11139.711,E2 -11139.711} C_VEL
LIN {X 0,Y 397.159,Z 256.512,A -85,B 0,C 180,E1 -11142.851,E2 -11142.851} C_VEL
LIN {X 0,Y 397.209,Z 256.506,A -85,B 0,C 180,E1 -11146.709,E2 -11146.709} C_VEL
LIN {X 0,Y 397.199,Z 256.505,A -85,B 0,C 180,E1 -11149.815,E2 -11149.815} C_VEL
LIN {X 0,Y 397.316,Z 256.496,A -85,B 0,C 180,E1 -11152.894,E2 -11152.894} C_VEL
LIN {X 0,Y 397.231,Z 256.507,A -85,B 0,C 180,E1 -11154.931,E2 -11154.931} C_VEL
LIN {X 0,Y 397.437,Z 256.475,A -85,B 0,C 180,E1 -11157.979,E2 -11157.979} C_VEL
LIN {X 0,Y 397.565,Z 256.459,A -85,B 0,C 180,E1 -11160.006,E2 -11160.006} C_VEL
LIN {X 0,Y 397.321,Z 256.492,A -85,B 0,C 180,E1 -11163.048,E2 -11163.048} C_VEL
LIN {X 0,Y 397.342,Z 256.488,A -85,B 0,C 180,E1 -11166.098,E2 -11166.098} C_VEL
LIN {X 0,Y 397.23,Z 256.501,A -85,B 0,C 180,E1 -11169.168,E2 -11169.168} C_VEL
LIN {X 0,Y 397.216,Z 256.507,A -85,B 0,C 180,E1 -11172.263,E2 -11172.263} C_VEL
LIN {X 0,Y 397.178,Z 256.507,A -85,B 0,C 180,E1 -11175.397,E2 -11175.397} C_VEL
LIN {X 0,Y 397.158,Z 256.513,A -85,B 0,C 180,E1 -11178.579,E2 -11178.579} C_VEL
LIN {X 0,Y 397.098,Z 256.519,A -85,B 0,C 180,E1 -11181.823,E2 -11181.823} C_VEL
LIN {X 0,Y 397.111,Z 256.515,A -85,B 0,C 180,E1 -11185.14,E2 -11185.14} C_VEL
LIN {X 0,Y 397.08,Z 256.521,A -85,B 0,C 180,E1 -11188.552,E2 -11188.552} C_VEL
LIN {X 0,Y 397.088,Z 256.524,A -85,B 0,C 180,E1 -11191.84,E2 -11191.84} C_VEL
LIN {X 0,Y 397.127,Z 256.518,A -85,B 0,C 180,E1 -11194.498,E2 -11194.498} C_VEL
LIN {X 0,Y 397.102,Z 256.523,A -85,B 0,C 180,E1 -11198.28,E2 -11198.28} C_VEL
LIN {X 0,Y 397.328,Z 258.174,A -85,B 0,C 180,E1 -11200.485,E2 -11200.485} C_VEL
LIN {X 0,Y 397.76,Z 261.07,A -85,B 0,C 180,E1 -11203.58,E2 -11203.58} C_VEL
LIN {X 0,Y 398.067,Z 264.027,A -85,B 0,C 180,E1 -11206.485,E2 -11206.485} C_VEL
LIN {X 0,Y 398.011,Z 267.256,A -85,B 0,C 180,E1 -11209.406,E2 -11209.406} C_VEL
LIN {X 0,Y 397.733,Z 271.167,A -85,B 0,C 180,E1 -11212.675,E2 -11212.675} C_VEL
LIN {X 0,Y 397.344,Z 275.681,A -85,B 0,C 180,E1 -11216.239,E2 -11216.239} C_VEL
LIN {X 0,Y 397.006,Z 279.525,A -85,B 0,C 180,E1 -11219.112,E2 -11219.112} C_VEL
LIN {X 0,Y 396.586,Z 284.352,A -85,B 0,C 180,E1 -11222.565,E2 -11222.565} C_VEL
LIN {X 0,Y 396.284,Z 289.226,A -85,B 0,C 180,E1 -11225.928,E2 -11225.928} C_VEL
LIN {X 0,Y 396.071,Z 294.151,A -85,B 0,C 180,E1 -11229.214,E2 -11229.214} C_VEL
LIN {X 0,Y 395.913,Z 298.037,A -85,B 0,C 180,E1 -11231.796,E2 -11231.796} C_VEL
LIN {X 0,Y 398.04,Z 308.625,A -85,B 0,C 180,E1 -11232.235,E2 -11232.235} C_VEL
LIN {X 0,Y 399.713,Z 318.488,A -85,B 0,C 180,E1 -11232.756,E2 -11232.756} C_VEL
LIN {X 0,Y 400.769,Z 327.2,A -85,B 0,C 180,E1 -11233.306,E2 -11233.306} C_VEL
LIN {X 0,Y 400.572,Z 334.809,A -85,B 0,C 180,E1 -11233.828,E2 -11233.828} C_VEL
LIN {X 0,Y 399.847,Z 344.085,A -85,B 0,C 180,E1 -11234.583,E2 -11234.583} C_VEL
LIN {X 0,Y 399.111,Z 353.035,A -85,B 0,C 180,E1 -11235.468,E2 -11235.468} C_VEL
LIN {X 0,Y 398.554,Z 359.989,A -85,B 0,C 180,E1 -11236.276,E2 -11236.276} C_VEL
LIN {X 0,Y 397.866,Z 368.783,A -85,B 0,C 180,E1 -11237.503,E2 -11237.503} C_VEL
LIN {X 0,Y 397.299,Z 374.985,A -85,B 0,C 180,E1 -11238.521,E2 -11238.521} C_VEL
LIN {X 0,Y 396.809,Z 381.524,A -85,B 0,C 180,E1 -11239.799,E2 -11239.799} C_VEL
LIN {X 0,Y 396.429,Z 386.024,A -85,B 0,C 180,E1 -11240.819,E2 -11240.819} C_VEL
LIN {X 0,Y 396.086,Z 391.516,A -85,B 0,C 180,E1 -11242.353,E2 -11242.353} C_VEL
LIN {X 0,Y 395.877,Z 395.84,A -85,B 0,C 180,E1 -11243.886,E2 -11243.886} C_VEL
LIN {X 0,Y 395.851,Z 398.208,A -85,B 0,C 180,E1 -11244.907,E2 -11244.907} C_VEL
LIN {X 0,Y 395.772,Z 400.005,A -85,B 0,C 180,E1 -11245.927,E2 -11245.927} C_VEL
LIN {X 0,Y 395.767,Z 402.45,A -85,B 0,C 180,E1 -11247.965,E2 -11247.965} C_VEL
LIN {X 0,Y 395.784,Z 403.038,A -85,B 0,C 180,E1 -11248.983,E2 -11248.983} C_VEL
LIN {X 0,Y 395.784,Z 403.038,A -85,B 0,C 180,E1 -11251.017,E2 -11251.017} C_VEL
LIN {X 0,Y 395.767,Z 402.45,A -85,B 0,C 180,E1 -11252.035,E2 -11252.035} C_VEL
LIN {X 0,Y 395.772,Z 400.005,A -85,B 0,C 180,E1 -11254.073,E2 -11254.073} C_VEL
LIN {X 0,Y 395.851,Z 398.208,A -85,B 0,C 180,E1 -11255.093,E2 -11255.093} C_VEL
LIN {X 0,Y 395.934,Z 394.602,A -85,B 0,C 180,E1 -11256.625,E2 -11256.625} C_VEL
LIN {X 0,Y 396.2,Z 389.856,A -85,B 0,C 180,E1 -11258.158,E2 -11258.158} C_VEL
LIN {X 0,Y 396.616,Z 383.835,A -85,B 0,C 180,E1 -11259.691,E2 -11259.691} C_VEL
LIN {X 0,Y 397.055,Z 377.737,A -85,B 0,C 180,E1 -11260.969,E2 -11260.969} C_VEL
LIN {X 0,Y 397.59,Z 372.038,A -85,B 0,C 180,E1 -11261.987,E2 -11261.987} C_VEL
LIN {X 0,Y 398.286,Z 363.482,A -85,B 0,C 180,E1 -11263.261,E2 -11263.261} C_VEL
LIN {X 0,Y 398.921,Z 355.3,A -85,B 0,C 180,E1 -11264.279,E2 -11264.279} C_VEL
LIN {X 0,Y 399.572,Z 346.923,A -85,B 0,C 180,E1 -11265.154,E2 -11265.154} C_VEL
LIN {X 0,Y 400.246,Z 338.071,A -85,B 0,C 180,E1 -11265.924,E2 -11265.924} C_VEL
LIN {X 0,Y 400.899,Z 328.743,A -85,B 0,C 180,E1 -11266.588,E2 -11266.588} C_VEL
LIN {X 0,Y 399.712,Z 318.494,A -85,B 0,C 180,E1 -11267.243,E2 -11267.243} C_VEL
LIN {X 0,Y 397.997,Z 308.261,A -85,B 0,C 180,E1 -11267.78,E2 -11267.78} C_VEL
LIN {X 0,Y 395.916,Z 298.003,A -85,B 0,C 180,E1 -11268.228,E2 -11268.228} C_VEL
LIN {X 0,Y 396.071,Z 294.133,A -85,B 0,C 180,E1 -11270.786,E2 -11270.786} C_VEL
LIN {X 0,Y 396.287,Z 289.214,A -85,B 0,C 180,E1 -11274.072,E2 -11274.072} C_VEL
LIN {X 0,Y 396.596,Z 284.083,A -85,B 0,C 180,E1 -11277.614,E2 -11277.614} C_VEL
LIN {X 0,Y 397.009,Z 279.517,A -85,B 0,C 180,E1 -11280.888,E2 -11280.888} C_VEL
LIN {X 0,Y 397.345,Z 275.677,A -85,B 0,C 180,E1 -11283.761,E2 -11283.761} C_VEL
LIN {X 0,Y 397.725,Z 271.14,A -85,B 0,C 180,E1 -11287.323,E2 -11287.323} C_VEL
LIN {X 0,Y 398.032,Z 267.023,A -85,B 0,C 180,E1 -11290.79,E2 -11290.79} C_VEL
LIN {X 0,Y 398.062,Z 263.9,A -85,B 0,C 180,E1 -11293.62,E2 -11293.62} C_VEL
LIN {X 0,Y 397.763,Z 261.034,A -85,B 0,C 180,E1 -11296.438,E2 -11296.438} C_VEL
LIN {X 0,Y 397.226,Z 257.365,A -85,B 0,C 180,E1 -11300.431,E2 -11300.431} C_VEL
LIN {X 0,Y 397.102,Z 256.522,A -85,B 0,C 180,E1 -11301.72,E2 -11301.72} C_VEL
LIN {X 0,Y 397.127,Z 256.521,A -85,B 0,C 180,E1 -11305.502,E2 -11305.502} C_VEL
LIN {X 0,Y 397.083,Z 256.519,A -85,B 0,C 180,E1 -11309.113,E2 -11309.113} C_VEL
LIN {X 0,Y 397.099,Z 256.517,A -85,B 0,C 180,E1 -11312.598,E2 -11312.598} C_VEL
LIN {X 0,Y 397.124,Z 256.519,A -85,B 0,C 180,E1 -11315.976,E2 -11315.976} C_VEL
LIN {X 0,Y 397.142,Z 256.518,A -85,B 0,C 180,E1 -11319.7,E2 -11319.7} C_VEL
LIN {X 0,Y 397.183,Z 256.507,A -85,B 0,C 180,E1 -11322.84,E2 -11322.84} C_VEL
LIN {X 0,Y 397.228,Z 256.501,A -85,B 0,C 180,E1 -11326.697,E2 -11326.697} C_VEL
LIN {X 0,Y 397.21,Z 256.506,A -85,B 0,C 180,E1 -11329.803,E2 -11329.803} C_VEL
LIN {X 0,Y 397.325,Z 256.49,A -85,B 0,C 180,E1 -11332.882,E2 -11332.882} C_VEL
LIN {X 0,Y 397.233,Z 256.502,A -85,B 0,C 180,E1 -11334.919,E2 -11334.919} C_VEL
LIN {X 0,Y 397.432,Z 256.476,A -85,B 0,C 180,E1 -11337.967,E2 -11337.967} C_VEL
LIN {X 0,Y 397.565,Z 256.459,A -85,B 0,C 180,E1 -11339.994,E2 -11339.994} C_VEL
LIN {X 0,Y 397.36,Z 256.49,A -85,B 0,C 180,E1 -11343.035,E2 -11343.035} C_VEL
LIN {X 0,Y 397.316,Z 256.496,A -85,B 0,C 180,E1 -11347.106,E2 -11347.106} C_VEL
LIN {X 0,Y 397.199,Z 256.505,A -85,B 0,C 180,E1 -11350.185,E2 -11350.185} C_VEL
LIN {X 0,Y 397.207,Z 256.506,A -85,B 0,C 180,E1 -11353.315,E2 -11353.315} C_VEL
LIN {X 0,Y 397.159,Z 256.512,A -85,B 0,C 180,E1 -11357.149,E2 -11357.149} C_VEL
LIN {X 0,Y 397.076,Z 256.527,A -85,B 0,C 180,E1 -11360.724,E2 -11360.724} C_VEL
LIN {X 0,Y 397.1,Z 256.518,A -85,B 0,C 180,E1 -11364.012,E2 -11364.012} C_VEL
LIN {X 0,Y 397.162,Z 256.509,A -85,B 0,C 180,E1 -11367.384,E2 -11367.384} C_VEL
LIN {X 0,Y 397.043,Z 256.526,A -85,B 0,C 180,E1 -11370.877,E2 -11370.877} C_VEL
LIN {X 0,Y 397.088,Z 256.524,A -85,B 0,C 180,E1 -11374.487,E2 -11374.487} C_VEL
LIN {X 0,Y 397.068,Z 256.528,A -85,B 0,C 180,E1 -11378.269,E2 -11378.269} C_VEL
LIN {X 0,Y 397.113,Z 256.52,A -85,B 0,C 180,E1 -11381.988,E2 -11381.988} C_VEL
LIN {X 0,Y 397.107,Z 256.516,A -85,B 0,C 180,E1 -11385.054,E2 -11385.054} C_VEL
LIN {X 0,Y 397.108,Z 256.522,A -85,B 0,C 180,E1 -11388.002,E2 -11388.002} C_VEL
LIN {X 0,Y 397.059,Z 256.526,A -85,B 0,C 180,E1 -11391.721,E2 -11391.721} C_VEL
LIN {X 0,Y 397.071,Z 256.523,A -85,B 0,C 180,E1 -11395.502,E2 -11395.502} C_VEL
LIN {X 0,Y 397.027,Z 256.527,A -85,B 0,C 180,E1 -11399.114,E2 -11399.114} C_VEL
LIN {X 0,Y 397.137,Z 256.512,A -85,B 0,C 180,E1 -11402.606,E2 -11402.606} C_VEL
LIN {X 0,Y 397.082,Z 256.522,A -85,B 0,C 180,E1 -11405.979,E2 -11405.979} C_VEL
LIN {X 0,Y 397.097,Z 256.521,A -85,B 0,C 180,E1 -11409.27,E2 -11409.27} C_VEL
LIN {X 0,Y 397.122,Z 256.519,A -85,B 0,C 180,E1 -11412.842,E2 -11412.842} C_VEL
LIN {X 0,Y 397.123,Z 256.52,A -85,B 0,C 180,E1 -11415.655,E2 -11415.655} C_VEL
LIN {X 0,Y 397.149,Z 256.516,A -85,B 0,C 180,E1 -11418.776,E2 -11418.776} C_VEL
LIN {X 0,Y 397.335,Z 256.492,A -85,B 0,C 180,E1 -11422.036,E2 -11422.036} C_VEL
LIN {X 0,Y 397.334,Z 256.493,A -85,B 0,C 180,E1 -11423.908,E2 -11423.908} C_VEL
LIN {X 0,Y 397.388,Z 256.485,A -85,B 0,C 180,E1 -11427.973,E2 -11427.973} C_VEL
LIN {X 0,Y 397.518,Z 256.471,A -85,B 0,C 180,E1 -11430,E2 -11430} C_VEL
LIN {X 0,Y 397.325,Z 256.493,A -85,B 0,C 180,E1 -11433.042,E2 -11433.042} C_VEL
LIN {X 0,Y 397.328,Z 256.493,A -85,B 0,C 180,E1 -11437.112,E2 -11437.112} C_VEL
LIN {X 0,Y 397.169,Z 256.514,A -85,B 0,C 180,E1 -11440.192,E2 -11440.192} C_VEL
LIN {X 0,Y 397.164,Z 256.514,A -85,B 0,C 180,E1 -11443.323,E2 -11443.323} C_VEL
LIN {X 0,Y 397.11,Z 256.522,A -85,B 0,C 180,E1 -11446.449,E2 -11446.449} C_VEL
LIN {X 0,Y 397.114,Z 256.518,A -85,B 0,C 180,E1 -11449.648,E2 -11449.648} C_VEL
LIN {X 0,Y 397.116,Z 256.516,A -85,B 0,C 180,E1 -11453.057,E2 -11453.057} C_VEL
LIN {X 0,Y 397.077,Z 256.525,A -85,B 0,C 180,E1 -11456.299,E2 -11456.299} C_VEL
LIN {X 0,Y 396.406,Z 256.604,A -85,B 0,C 180,E1 -11457.146,E2 -11457.146} C_VEL
LIN {X 0,Y 393.536,Z 256.965,A -85,B 0,C 180,E1 -11458.522,E2 -11458.522} C_VEL
LIN {X 0,Y 391.101,Z 257.27,A -85,B 0,C 180,E1 -11459.634,E2 -11459.634} C_VEL
LIN {X 0,Y 390.049,Z 257.399,A -85,B 0,C 180,E1 -11460.494,E2 -11460.494} C_VEL
LIN {X 0,Y 389.96,Z 257.408,A -85,B 0,C 180,E1 -11460.785,E2 -11460.785} C_VEL
LIN {X 0,Y 390.015,Z 257.405,A -85,B 0,C 180,E1 -11464.029,E2 -11464.029} C_VEL
LIN {X 0,Y 389.996,Z 257.403,A -85,B 0,C 180,E1 -11467.556,E2 -11467.556} C_VEL
LIN {X 0,Y 390.034,Z 257.397,A -85,B 0,C 180,E1 -11470.831,E2 -11470.831} C_VEL
LIN {X 0,Y 390.083,Z 257.398,A -85,B 0,C 180,E1 -11473.903,E2 -11473.903} C_VEL
LIN {X 0,Y 390.074,Z 257.392,A -85,B 0,C 180,E1 -11476.804,E2 -11476.804} C_VEL
LIN {X 0,Y 390.035,Z 257.401,A -85,B 0,C 180,E1 -11479.569,E2 -11479.569} C_VEL
LIN {X 0,Y 390.006,Z 257.401,A -85,B 0,C 180,E1 -11482.455,E2 -11482.455} C_VEL
LIN {X 0,Y 390.031,Z 257.399,A -85,B 0,C 180,E1 -11486.051,E2 -11486.051} C_VEL
LIN {X 0,Y 390.011,Z 257.403,A -85,B 0,C 180,E1 -11489.876,E2 -11489.876} C_VEL
LIN {X 0,Y 390.082,Z 257.396,A -85,B 0,C 180,E1 -11493.238,E2 -11493.238} C_VEL
LIN {X 0,Y 390.04,Z 257.398,A -85,B 0,C 180,E1 -11496.77,E2 -11496.77} C_VEL
LIN {X 0,Y 390.078,Z 257.392,A -85,B 0,C 180,E1 -11499.989,E2 -11499.989} C_VEL
LIN {X 0,Y 390.115,Z 257.393,A -85,B 0,C 180,E1 -11503.255,E2 -11503.255} C_VEL
LIN {X 0,Y 390.175,Z 257.381,A -85,B 0,C 180,E1 -11506.568,E2 -11506.568} C_VEL
LIN {X 0,Y 390.149,Z 257.384,A -85,B 0,C 180,E1 -11509.629,E2 -11509.629} C_VEL
LIN {X 0,Y 390.264,Z 257.373,A -85,B 0,C 180,E1 -11512.765,E2 -11512.765} C_VEL
LIN {X 0,Y 390.202,Z 257.382,A -85,B 0,C 180,E1 -11514.84,E2 -11514.84} C_VEL
LIN {X 0,Y 390.406,Z 257.351,A -85,B 0,C 180,E1 -11517.943,E2 -11517.943} C_VEL
LIN {X 0,Y 390.535,Z 257.335,A -85,B 0,C 180,E1 -11520.006,E2 -11520.006} C_VEL
LIN {X 0,Y 390.258,Z 257.371,A -85,B 0,C 180,E1 -11523.103,E2 -11523.103} C_VEL
LIN {X 0,Y 390.297,Z 257.367,A -85,B 0,C 180,E1 -11526.208,E2 -11526.208} C_VEL
LIN {X 0,Y 390.188,Z 257.378,A -85,B 0,C 180,E1 -11529.335,E2 -11529.335} C_VEL
LIN {X 0,Y 390.168,Z 257.387,A -85,B 0,C 180,E1 -11532.489,E2 -11532.489} C_VEL
LIN {X 0,Y 390.138,Z 257.385,A -85,B 0,C 180,E1 -11535.682,E2 -11535.682} C_VEL
LIN {X 0,Y 390.103,Z 257.389,A -85,B 0,C 180,E1 -11538.927,E2 -11538.927} C_VEL
LIN {X 0,Y 390.04,Z 257.403,A -85,B 0,C 180,E1 -11542.239,E2 -11542.239} C_VEL
LIN {X 0,Y 390.055,Z 257.397,A -85,B 0,C 180,E1 -11545.727,E2 -11545.727} C_VEL
LIN {X 0,Y 390.036,Z 257.397,A -85,B 0,C 180,E1 -11549.116,E2 -11549.116} C_VEL
LIN {X 0,Y 390.049,Z 257.395,A -85,B 0,C 180,E1 -11552.726,E2 -11552.726} C_VEL
LIN {X 0,Y 390.052,Z 257.401,A -85,B 0,C 180,E1 -11555.826,E2 -11555.826} C_VEL
LIN {X 0,Y 390.047,Z 257.402,A -85,B 0,C 180,E1 -11557.784,E2 -11557.784} C_VEL
LIN {X 0,Y 390.181,Z 258.225,A -85,B 0,C 180,E1 -11559.24,E2 -11559.24} C_VEL
LIN {X 0,Y 390.579,Z 261.096,A -85,B 0,C 180,E1 -11562.462,E2 -11562.462} C_VEL
LIN {X 0,Y 390.94,Z 264.03,A -85,B 0,C 180,E1 -11565.485,E2 -11565.485} C_VEL
LIN {X 0,Y 391.02,Z 267.022,A -85,B 0,C 180,E1 -11568.317,E2 -11568.317} C_VEL
LIN {X 0,Y 390.843,Z 270.072,A -85,B 0,C 180,E1 -11570.998,E2 -11570.998} C_VEL
LIN {X 0,Y 390.506,Z 273.803,A -85,B 0,C 180,E1 -11574.089,E2 -11574.089} C_VEL
LIN {X 0,Y 390.146,Z 277.862,A -85,B 0,C 180,E1 -11577.289,E2 -11577.289} C_VEL
LIN {X 0,Y 389.691,Z 282.645,A -85,B 0,C 180,E1 -11580.861,E2 -11580.861} C_VEL
LIN {X 0,Y 389.335,Z 287.727,A -85,B 0,C 180,E1 -11584.504,E2 -11584.504} C_VEL
LIN {X 0,Y 389.104,Z 292.357,A -85,B 0,C 180,E1 -11587.71,E2 -11587.71} C_VEL
LIN {X 0,Y 388.866,Z 297.26,A -85,B 0,C 180,E1 -11591.016,E2 -11591.016} C_VEL
LIN {X 0,Y 388.858,Z 298.038,A -85,B 0,C 180,E1 -11591.46,E2 -11591.46} C_VEL
LIN {X 0,Y 391.058,Z 308.725,A -85,B 0,C 180,E1 -11591.919,E2 -11591.919} C_VEL
LIN {X 0,Y 392.831,Z 319.367,A -85,B 0,C 180,E1 -11592.501,E2 -11592.501} C_VEL
LIN {X 0,Y 393.944,Z 328.798,A -85,B 0,C 180,E1 -11593.127,E2 -11593.127} C_VEL
LIN {X 0,Y 393.62,Z 336.246,A -85,B 0,C 180,E1 -11593.668,E2 -11593.668} C_VEL
LIN {X 0,Y 392.845,Z 345.241,A -85,B 0,C 180,E1 -11594.434,E2 -11594.434} C_VEL
LIN {X 0,Y 392.128,Z 353.97,A -85,B 0,C 180,E1 -11595.336,E2 -11595.336} C_VEL
LIN {X 0,Y 391.453,Z 361.728,A -85,B 0,C 180,E1 -11596.288,E2 -11596.288} C_VEL
LIN {X 0,Y 390.916,Z 368.588,A -85,B 0,C 180,E1 -11597.278,E2 -11597.278} C_VEL
LIN {X 0,Y 390.311,Z 374.789,A -85,B 0,C 180,E1 -11598.313,E2 -11598.313} C_VEL
LIN {X 0,Y 389.782,Z 381.328,A -85,B 0,C 180,E1 -11599.613,E2 -11599.613} C_VEL
LIN {X 0,Y 389.393,Z 385.829,A -85,B 0,C 180,E1 -11600.652,E2 -11600.652} C_VEL
LIN {X 0,Y 389.038,Z 391.321,A -85,B 0,C 180,E1 -11602.213,E2 -11602.213} C_VEL
LIN {X 0,Y 388.811,Z 395.646,A -85,B 0,C 180,E1 -11603.774,E2 -11603.774} C_VEL
LIN {X 0,Y 388.749,Z 398.012,A -85,B 0,C 180,E1 -11604.814,E2 -11604.814} C_VEL
LIN {X 0,Y 388.698,Z 399.811,A -85,B 0,C 180,E1 -11605.853,E2 -11605.853} C_VEL
LIN {X 0,Y 388.665,Z 402.255,A -85,B 0,C 180,E1 -11607.928,E2 -11607.928} C_VEL
LIN {X 0,Y 388.698,Z 402.844,A -85,B 0,C 180,E1 -11608.964,E2 -11608.964} C_VEL
LIN {X 0,Y 388.698,Z 402.844,A -85,B 0,C 180,E1 -11611.036,E2 -11611.036} C_VEL
LIN {X 0,Y 388.665,Z 402.255,A -85,B 0,C 180,E1 -11612.072,E2 -11612.072} C_VEL
LIN {X 0,Y 388.698,Z 399.811,A -85,B 0,C 180,E1 -11614.147,E2 -11614.147} C_VEL
LIN {X 0,Y 388.737,Z 396.77,A -85,B 0,C 180,E1 -11615.746,E2 -11615.746} C_VEL
LIN {X 0,Y 388.95,Z 392.875,A -85,B 0,C 180,E1 -11617.266,E2 -11617.266} C_VEL
LIN {X 0,Y 389.263,Z 387.745,A -85,B 0,C 180,E1 -11618.828,E2 -11618.828} C_VEL
LIN {X 0,Y 389.674,Z 382.483,A -85,B 0,C 180,E1 -11620.128,E2 -11620.128} C_VEL
LIN {X 0,Y 390.172,Z 376.165,A -85,B 0,C 180,E1 -11621.428,E2 -11621.428} C_VEL
LIN {X 0,Y 390.759,Z 370.215,A -85,B 0,C 180,E1 -11622.464,E2 -11622.464} C_VEL
LIN {X 0,Y 391.33,Z 363.286,A -85,B 0,C 180,E1 -11623.501,E2 -11623.501} C_VEL
LIN {X 0,Y 391.99,Z 355.104,A -85,B 0,C 180,E1 -11624.537,E2 -11624.537} C_VEL
LIN {X 0,Y 392.727,Z 346.593,A -85,B 0,C 180,E1 -11625.438,E2 -11625.438} C_VEL
LIN {X 0,Y 393.4,Z 337.876,A -85,B 0,C 180,E1 -11626.208,E2 -11626.208} C_VEL
LIN {X 0,Y 394.041,Z 330.257,A -85,B 0,C 180,E1 -11626.772,E2 -11626.772} C_VEL
LIN {X 0,Y 392.909,Z 319.746,A -85,B 0,C 180,E1 -11627.476,E2 -11627.476} C_VEL
LIN {X 0,Y 391.144,Z 309.039,A -85,B 0,C 180,E1 -11628.065,E2 -11628.065} C_VEL
LIN {X 0,Y 388.847,Z 297.839,A -85,B 0,C 180,E1 -11628.572,E2 -11628.572} C_VEL
LIN {X 0,Y 389.009,Z 293.985,A -85,B 0,C 180,E1 -11631.181,E2 -11631.181} C_VEL
LIN {X 0,Y 389.238,Z 289.072,A -85,B 0,C 180,E1 -11634.537,E2 -11634.537} C_VEL
LIN {X 0,Y 389.562,Z 284.237,A -85,B 0,C 180,E1 -11637.973,E2 -11637.973} C_VEL
LIN {X 0,Y 390.022,Z 279.445,A -85,B 0,C 180,E1 -11641.504,E2 -11641.504} C_VEL
LIN {X 0,Y 390.312,Z 276.096,A -85,B 0,C 180,E1 -11644.072,E2 -11644.072} C_VEL
LIN {X 0,Y 390.712,Z 271.593,A -85,B 0,C 180,E1 -11647.703,E2 -11647.703} C_VEL
LIN {X 0,Y 391.005,Z 267.797,A -85,B 0,C 180,E1 -11650.977,E2 -11650.977} C_VEL
LIN {X 0,Y 391.054,Z 265.509,A -85,B 0,C 180,E1 -11653.072,E2 -11653.072} C_VEL
LIN {X 0,Y 390.779,Z 262.55,A -85,B 0,C 180,E1 -11656.002,E2 -11656.002} C_VEL
LIN {X 0,Y 390.33,Z 259.24,A -85,B 0,C 180,E1 -11659.59,E2 -11659.59} C_VEL
LIN {X 0,Y 390.148,Z 258.099,A -85,B 0,C 180,E1 -11660.91,E2 -11660.91} C_VEL
LIN {X 0,Y 390.048,Z 257.402,A -85,B 0,C 180,E1 -11662.447,E2 -11662.447} C_VEL
LIN {X 0,Y 390.077,Z 257.399,A -85,B 0,C 180,E1 -11665.971,E2 -11665.971} C_VEL
LIN {X 0,Y 390.05,Z 257.4,A -85,B 0,C 180,E1 -11669.866,E2 -11669.866} C_VEL
LIN {X 0,Y 390.053,Z 257.395,A -85,B 0,C 180,E1 -11673.222,E2 -11673.222} C_VEL
LIN {X 0,Y 390.071,Z 257.392,A -85,B 0,C 180,E1 -11676.76,E2 -11676.76} C_VEL
LIN {X 0,Y 390.106,Z 257.392,A -85,B 0,C 180,E1 -11679.978,E2 -11679.978} C_VEL
LIN {X 0,Y 390.139,Z 257.386,A -85,B 0,C 180,E1 -11683.243,E2 -11683.243} C_VEL
LIN {X 0,Y 390.194,Z 257.377,A -85,B 0,C 180,E1 -11686.556,E2 -11686.556} C_VEL
LIN {X 0,Y 390.162,Z 257.386,A -85,B 0,C 180,E1 -11689.617,E2 -11689.617} C_VEL
LIN {X 0,Y 390.273,Z 257.368,A -85,B 0,C 180,E1 -11692.753,E2 -11692.753} C_VEL
LIN {X 0,Y 390.205,Z 257.377,A -85,B 0,C 180,E1 -11694.827,E2 -11694.827} C_VEL
LIN {X 0,Y 390.4,Z 257.352,A -85,B 0,C 180,E1 -11697.931,E2 -11697.931} C_VEL
LIN {X 0,Y 390.535,Z 257.335,A -85,B 0,C 180,E1 -11699.994,E2 -11699.994} C_VEL
LIN {X 0,Y 390.294,Z 257.371,A -85,B 0,C 180,E1 -11703.09,E2 -11703.09} C_VEL
LIN {X 0,Y 390.264,Z 257.368,A -85,B 0,C 180,E1 -11706.599,E2 -11706.599} C_VEL
LIN {X 0,Y 390.176,Z 257.382,A -85,B 0,C 180,E1 -11709.323,E2 -11709.323} C_VEL
LIN {X 0,Y 390.151,Z 257.384,A -85,B 0,C 180,E1 -11712.477,E2 -11712.477} C_VEL
LIN {X 0,Y 390.117,Z 257.387,A -85,B 0,C 180,E1 -11715.671,E2 -11715.671} C_VEL
